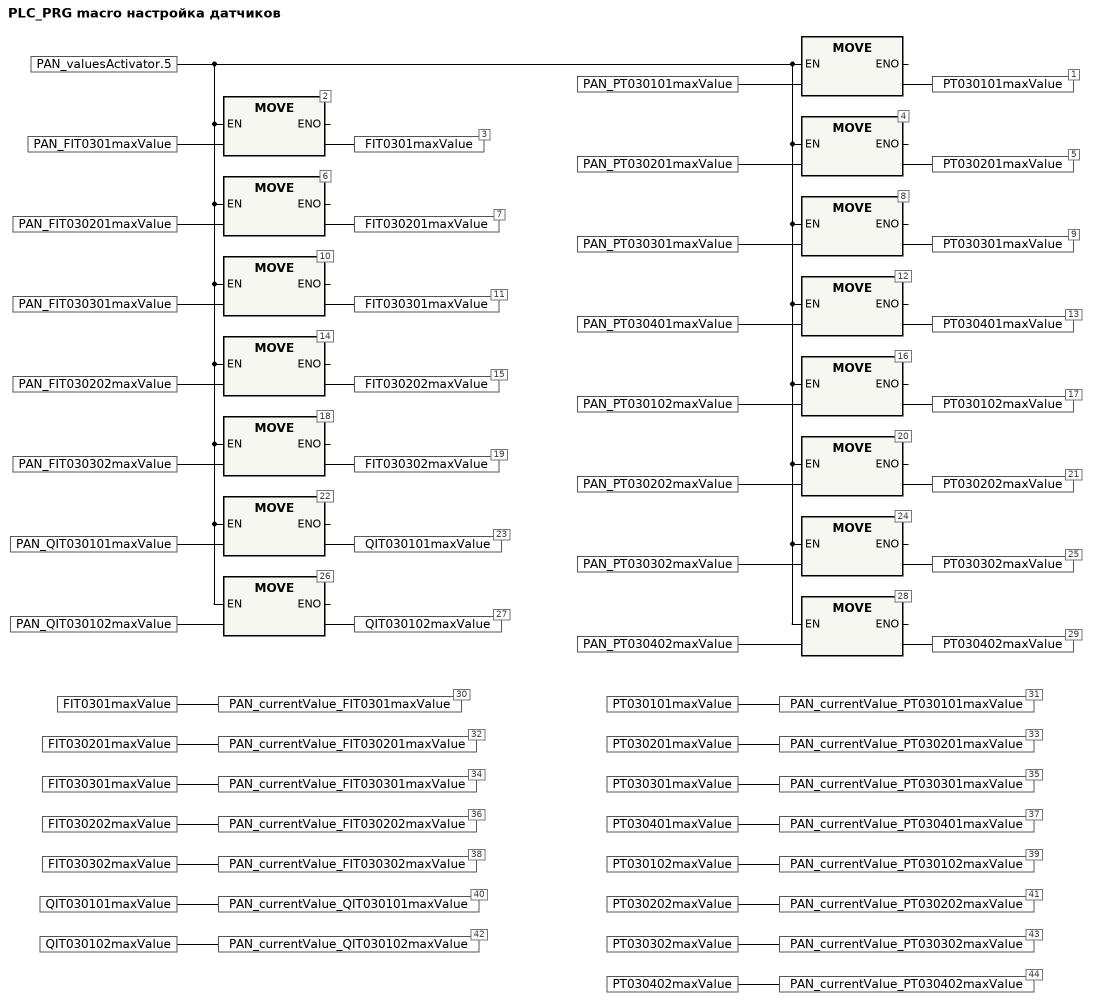
[picture p24: PLC_PRG macro настройка датчиков (CFC)]
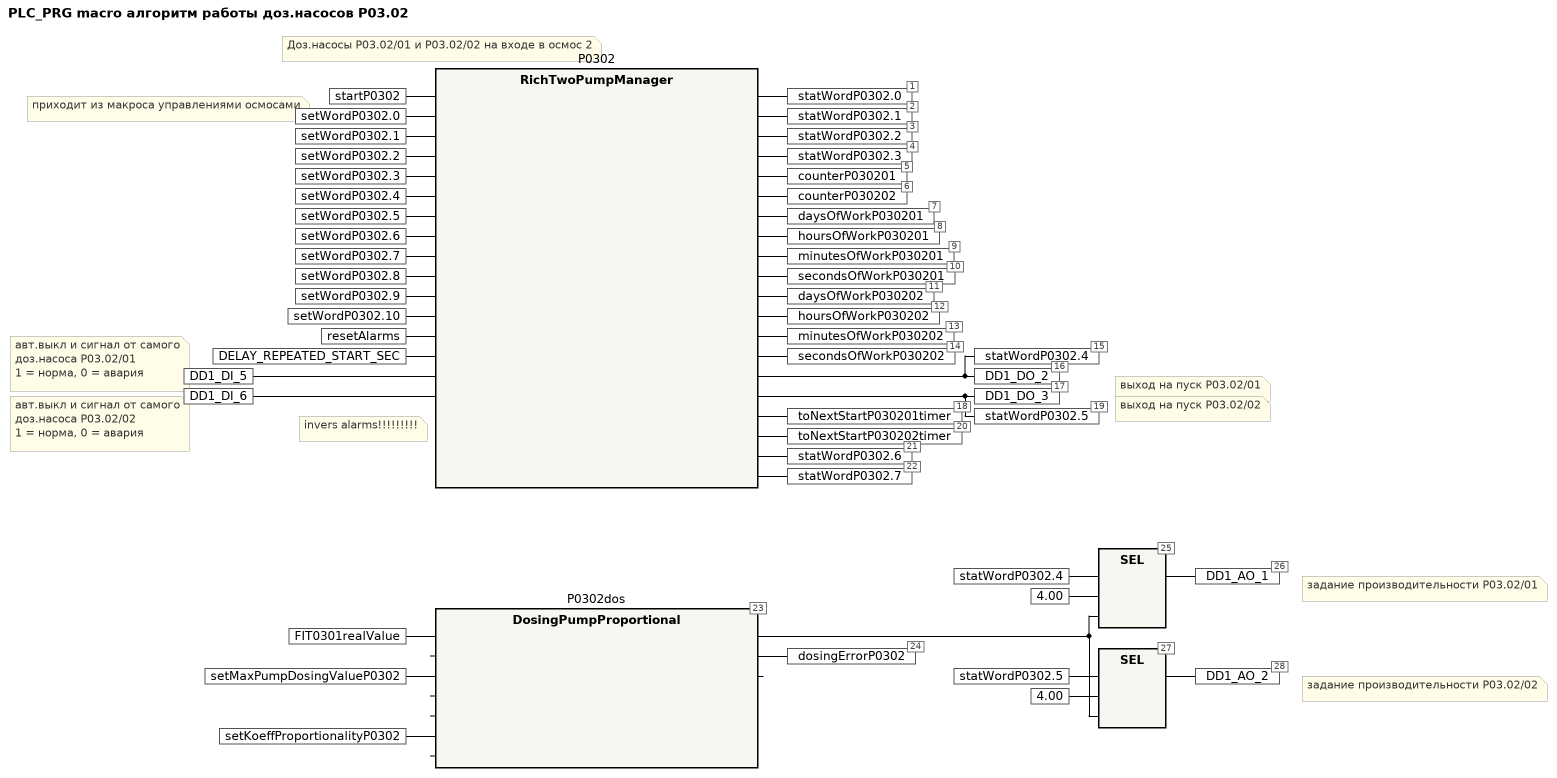
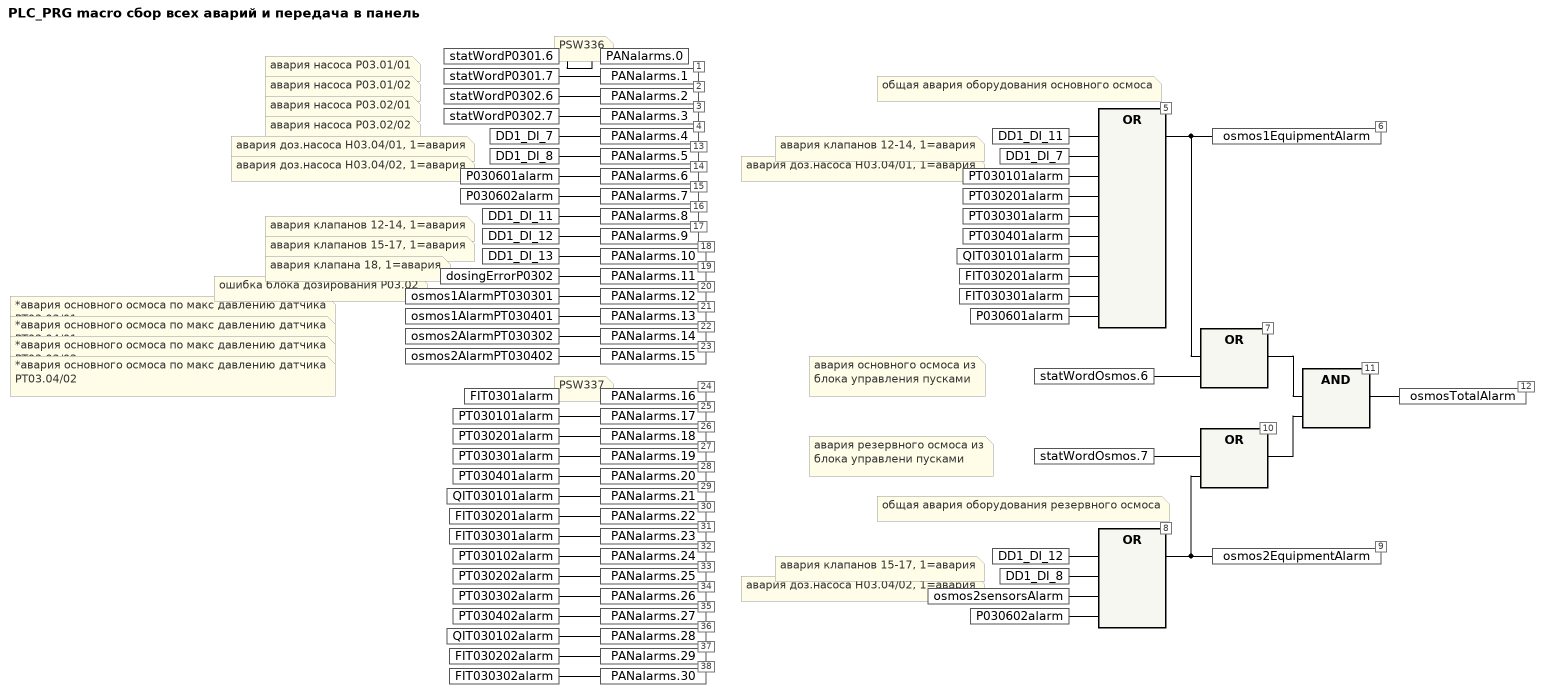
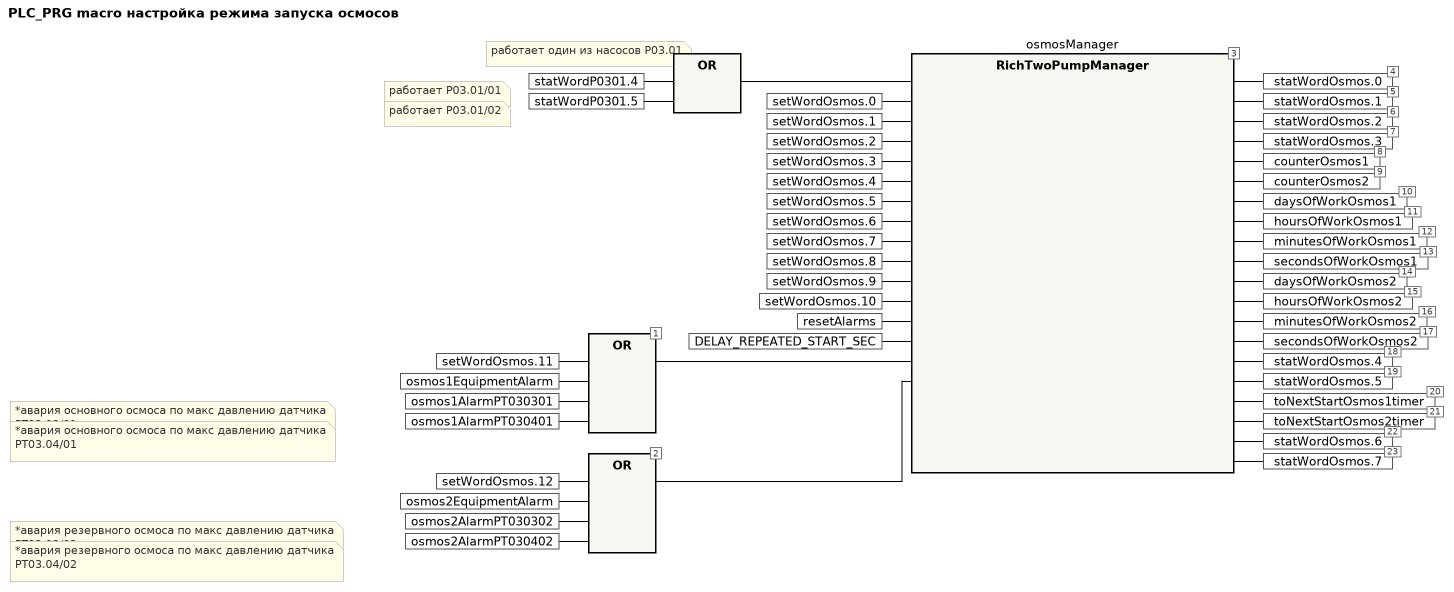
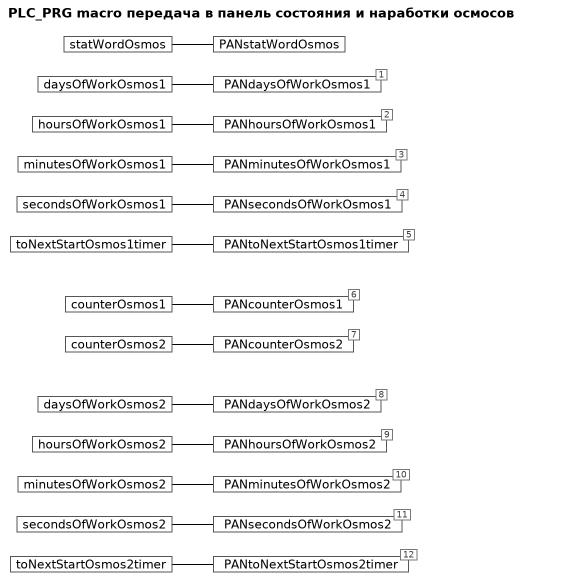
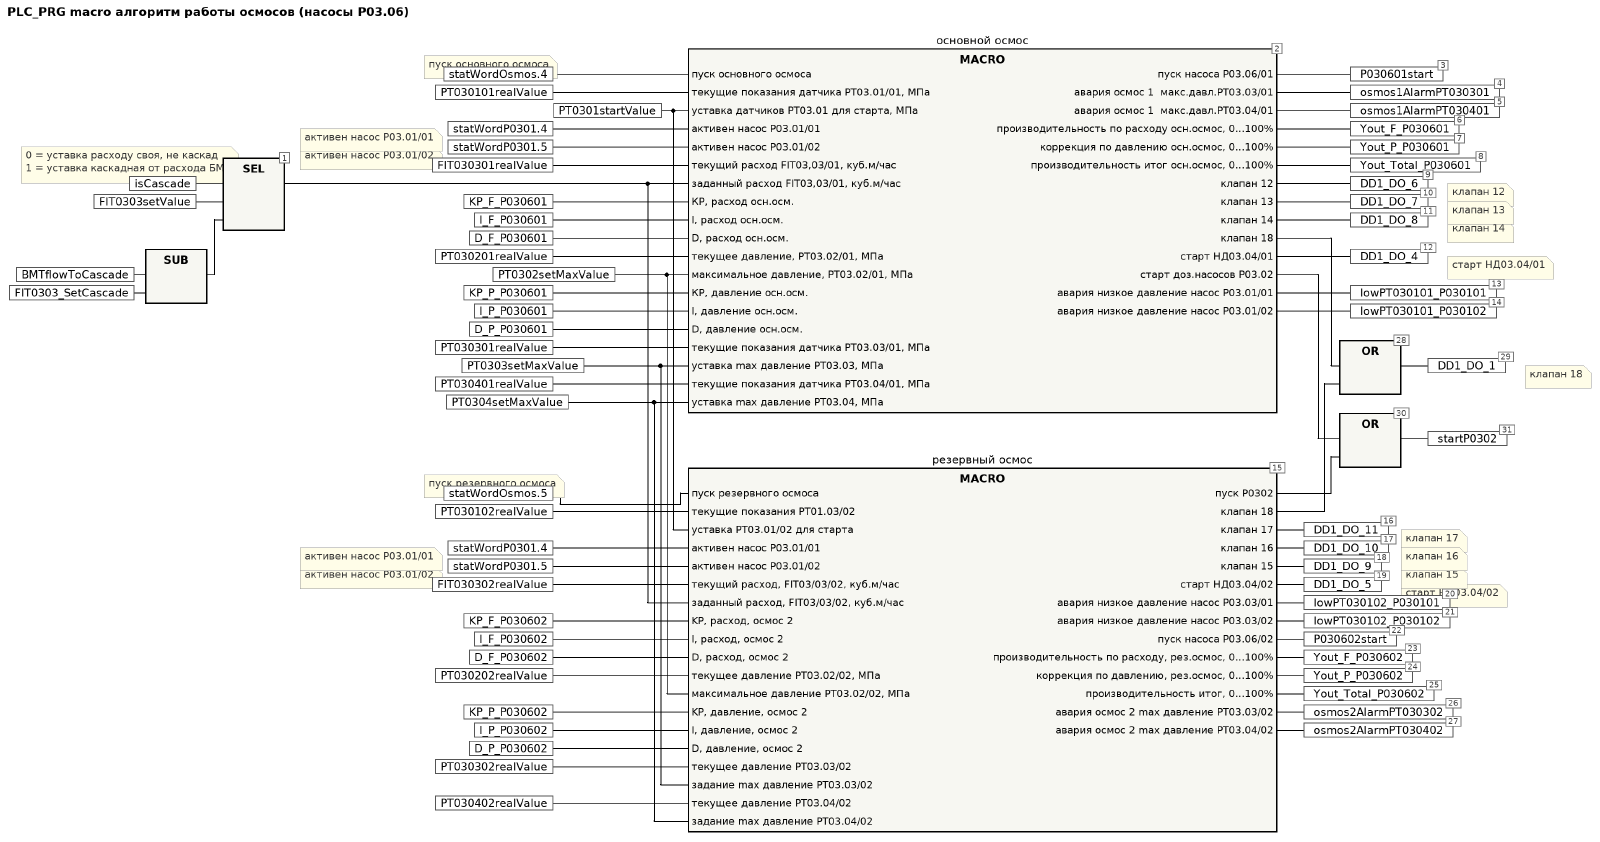
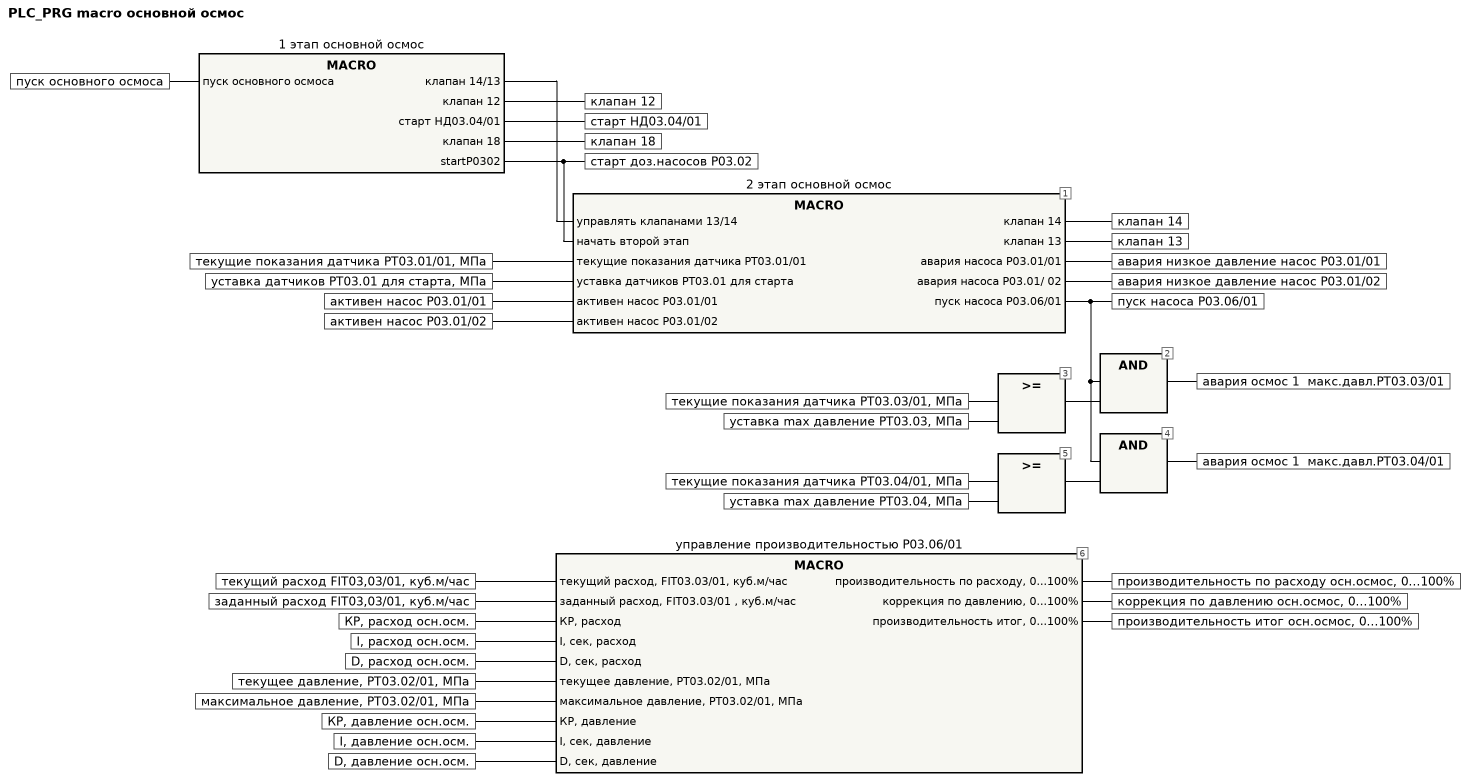
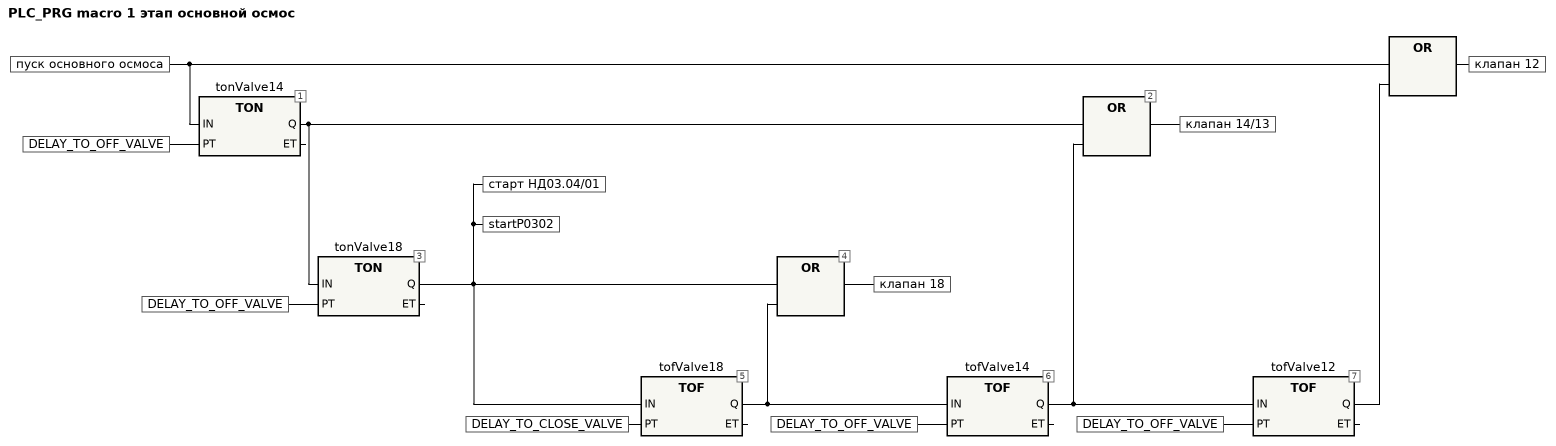
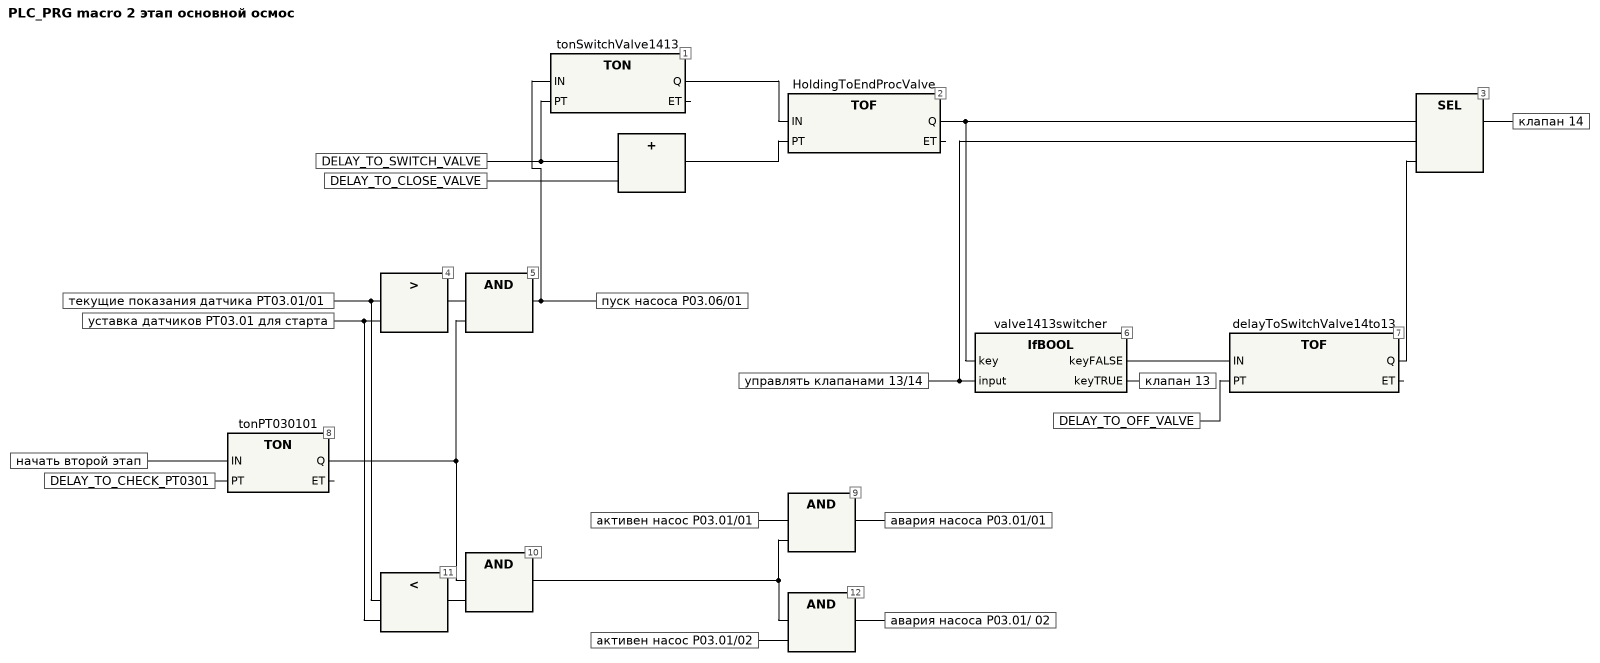
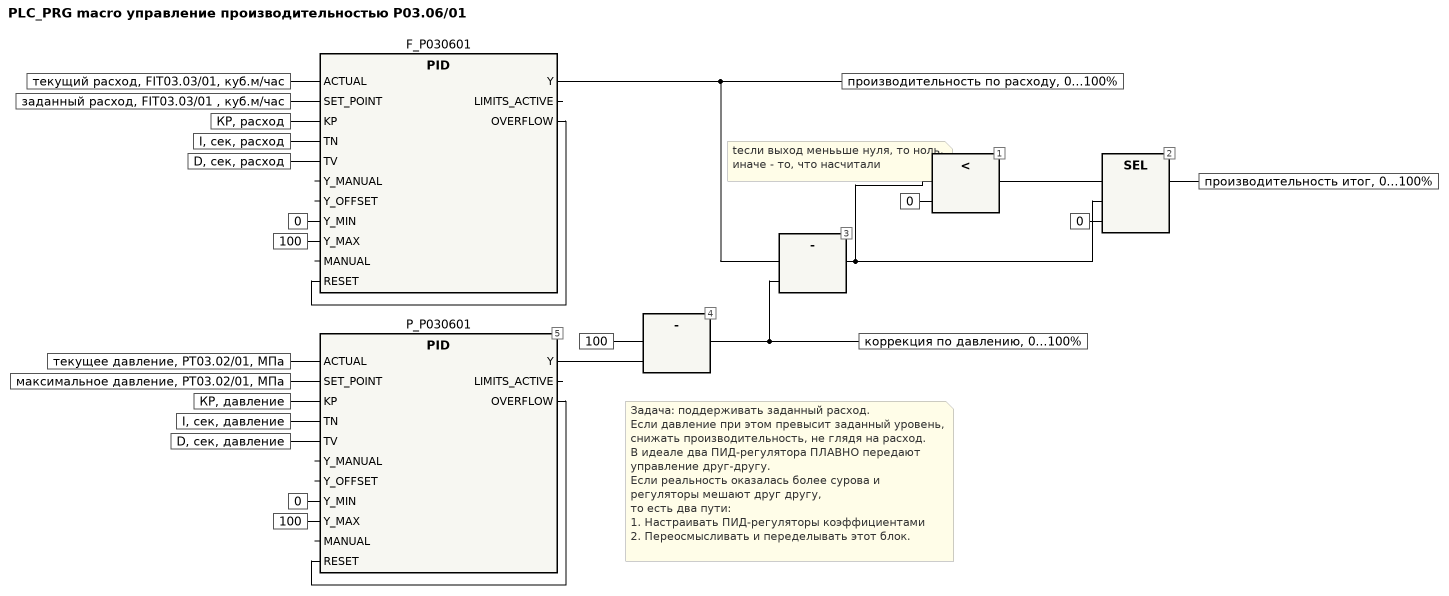
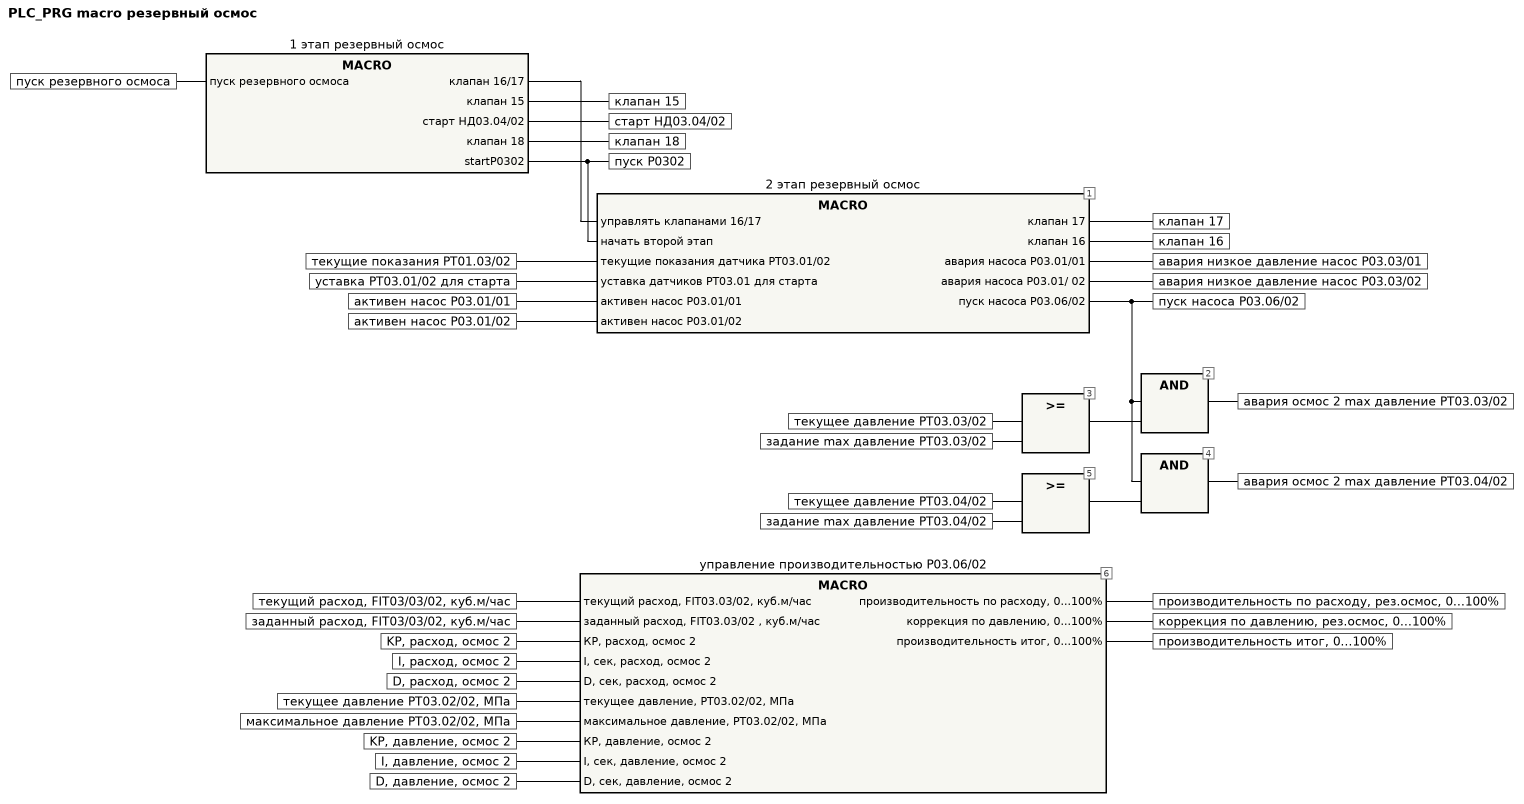
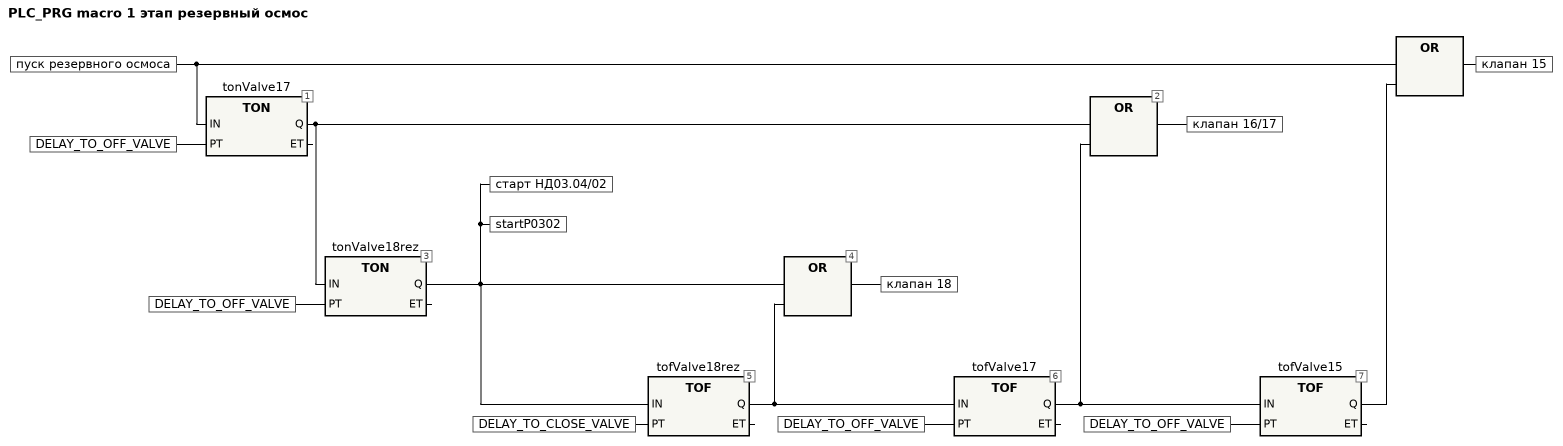
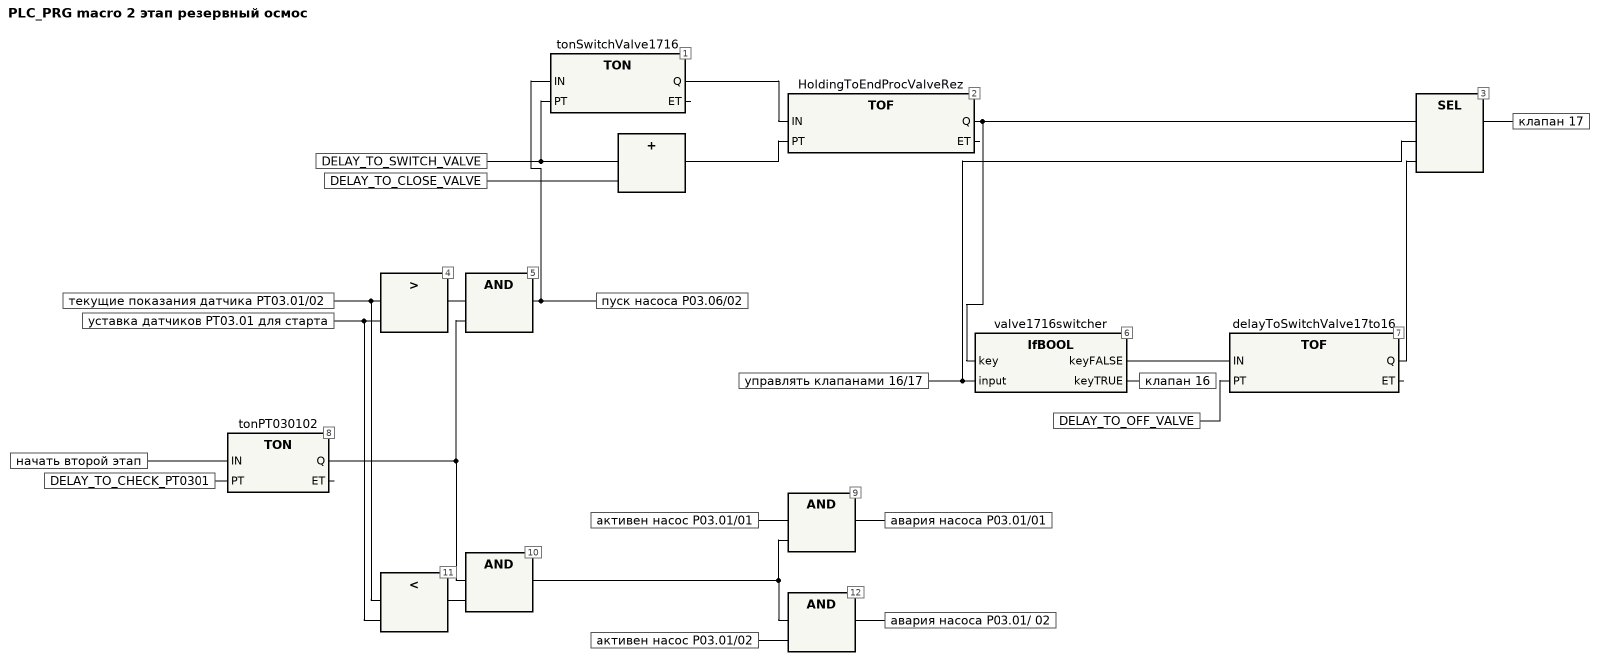
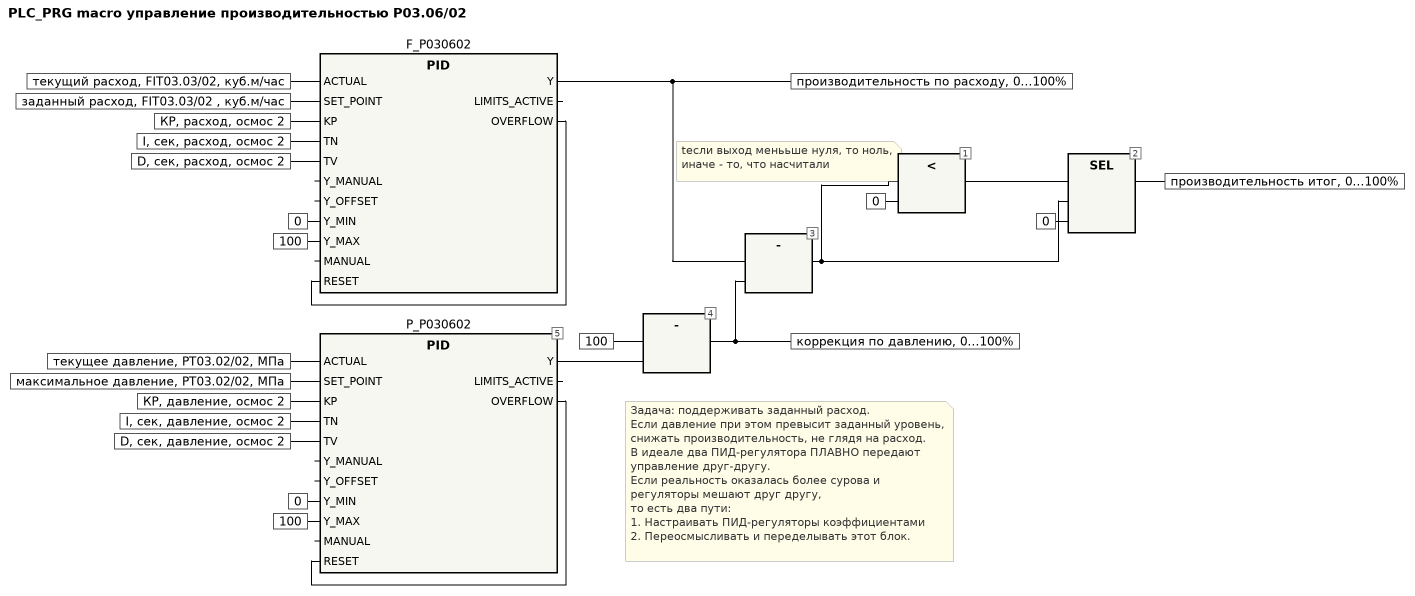
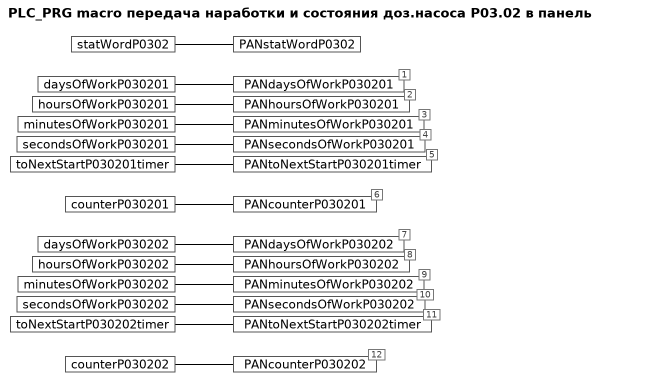
_CFC_ (* Continuous Function Chart, elements in execution order *)
(* восстановление заданного ранее режима / работы после подачи питания *)
(* командное слово удаленной панели *)
(* командное слово в локальной панели *)
(* - низкий уровень в емкости V02.07 / (сигнал из АСУ-2 осмос 1) 1 = true *)
(* - высокий уровень в емкости V06.01 / (сигнал из АСУ-1 общий) 1 = true *)
(* - высокий уровень в емкости V04.01 / (сигнал от БМТ, МЕ04) 1 = true *)
(* расход в БМТ для расчета каскадной уставки / получить из АСУ-1! *)
(* показ расхода БМТ в панели оператора *)
(* 0 = уставка расходу своя, не каскад / 1 = уставка каскадная от расхода БМТ *)
(* прием сигналов из разных источников / условие запуска см.в макросе "управление насосами Р03.01 *)
(* командное слово для осмоса *)
(* командное слово доз. насоса Р03.02 *)
(* командное слово насосов Р03.01 *)
(* PAN - переменные для панели в щите / OPAN - переменные для выносной панели, на установке *)
(* ******************добавь сюда вкл и выкл от выносной панели******************* / задание режима работы - каскад/не каскад *)
#0 onStartCatcher:R_TRIG(CLK: TRUE)
#1 OR(PANsetWordOsmos.11, #0.Q)
#2 resetAlarms <= #1
#3 setCascadeOnStart:IfBOOL(key: isCascadeOnStart, input: #0.Q)
#4 OR(#3.keyTRUE, PANsetWordOsmos.12)
#5 OR(#3.keyFALSE, PANsetWordOsmos.13)
#6 cascadeTrig:RS(SET: #4, RESET1: #5)
#7 statWordOsmos.8 <= #6.Q1
#8 isCascade <= #6.Q1
#9 MOVE(EN: #0.Q, setWordP0301onStart)
#10 setWordP0301 <= #9
#11 OR(#4, #5)
#12 MOVE(EN: #11, isCascade)
#13 isCascadeOnStart <= #12
#14 MOVE(EN: #0.Q, setWordP0302onStart)
#15 setWordP0302 <= #14
#16 MOVE(EN: #0.Q, setWordOsmosOnStart)
#17 setWordOsmos <= #16
#18 lowLevelV0207 <= ASU_Levels.0
#19 highLevelV0601 <= ASU_Levels.1
#20 highLevelV0401 <= ASU_Levels.2
#21 BMTflowToCascade <= ASU_FlowFromBMT
#22 PAN_BMT_Flow <= BMTflowToCascade
#23 MACRO настройка расхода, каскада и допустимых давлений осмоса()
	(* значение, вычитаемое из расхода БМТ / задается в панели, коэф.каскад *)
	(* предельно допустимые давления *)
	(* некаскадная уставка на поддержание расхода *)
	(* мин.давление для старта осмосов *)
	#24 MOVE(EN: PAN_valuesActivator.0, PAN_FIT0303_SetCascade)
	#25 FIT0303_SetCascade <= #24
	#26 MOVE(EN: PAN_valuesActivator.0, PAN_PT0301startValue)
	#27 PT0301startValue <= #26
	#28 MOVE(EN: PAN_valuesActivator.0, PAN_FIT0303setValue)
	#29 FIT0303setValue <= #28
	#30 MOVE(EN: PAN_valuesActivator.0, PAN_PT0302setMaxValue)
	#31 PT0302setMaxValue <= #30
	#32 MOVE(EN: PAN_valuesActivator.0, PAN_PT0303setMaxValue)
	#33 PT0303setMaxValue <= #32
	#34 MOVE(EN: PAN_valuesActivator.0, PAN_PT0304setMaxValue)
	#35 PT0304setMaxValue <= #34
	#36 PAN_currentValue_PT0301startValue <= PT0301startValue
	#37 PAN_currentValue_FIT0303setValue <= FIT0303setValue
	#38 PAN_currentValue_PT0302setMaxValue <= PT0302setMaxValue
	#39 PAN_currentValue_PT0303setMaxValue <= PT0303setMaxValue
	#40 PAN_currentValue_PT0304setMaxValue <= PT0304setMaxValue
	#41 PAN_currentValue_FIT0303_SetCascade <= FIT0303_SetCascade
END_MACRO
#42 MACRO коэффициенты ПИД-регуляторов осмосов()
	(* осмос 1 *)
	(* осмос 2 *)
	(* PID по расходу *)
	(* PID по давлению *)
	(* PID по расходу *)
	(* PID по давлению *)
	#43 MOVE(EN: PAN_valuesActivator.1, PAN_KP_F_P030601)
	#44 KP_F_P030601 <= #43
	#45 MOVE(EN: PAN_valuesActivator.1, PAN_I_F_P030601)
	#46 I_F_P030601 <= #45
	#47 MOVE(EN: PAN_valuesActivator.1, PAN_D_F_P030601)
	#48 D_F_P030601 <= #47
	#49 MOVE(EN: PAN_valuesActivator.1, PAN_KP_P_P030601)
	#50 KP_P_P030601 <= #49
	#51 MOVE(EN: PAN_valuesActivator.1, PAN_I_P_P030601)
	#52 I_P_P030601 <= #51
	#53 MOVE(EN: PAN_valuesActivator.1, PAN_D_P_P030601)
	#54 D_P_P030601 <= #53
	#55 MOVE(EN: PAN_valuesActivator.2, PAN_KP_F_P030602)
	#56 KP_F_P030602 <= #55
	#57 MOVE(EN: PAN_valuesActivator.2, PAN_I_F_P030602)
	#58 I_F_P030602 <= #57
	#59 MOVE(EN: PAN_valuesActivator.2, PAN_D_F_P030602)
	#60 D_F_P030602 <= #59
	#61 MOVE(EN: PAN_valuesActivator.2, PAN_KP_P_P030602)
	#62 KP_P_P030602 <= #61
	#63 MOVE(EN: PAN_valuesActivator.2, PAN_I_P_P030602)
	#64 I_P_P030602 <= #63
	#65 MOVE(EN: PAN_valuesActivator.2, PAN_D_P_P030602)
	#66 D_P_P030602 <= #65
	#67 PAN_currentValue_KP_F_P030601 <= KP_F_P030601
	#68 PAN_currentValue_KP_F_P030602 <= KP_F_P030602
	#69 PAN_currentValue_I_F_P030601 <= I_F_P030601
	#70 PAN_currentValue_I_F_P030602 <= I_F_P030602
	#71 PAN_currentValue_D_F_P030601 <= D_F_P030601
	#72 PAN_currentValue_D_F_P030602 <= D_F_P030602
	#73 PAN_currentValue_KP_P_P030601 <= KP_P_P030601
	#74 PAN_currentValue_KP_P_P030602 <= KP_P_P030602
	#75 PAN_currentValue_I_P_P030601 <= I_P_P030601
	#76 PAN_currentValue_I_P_P030602 <= I_P_P030602
	#77 PAN_currentValue_D_P_P030601 <= D_P_P030601
	#78 PAN_currentValue_D_P_P030602 <= D_P_P030602
END_MACRO
#79 MACRO обмен сигналами с DD2 (ПР102)()
	(* передача производительности / Р03.06/02 через модбас *)
	(* производительность доз.насоса Р03.06/02 / в процентах 0...100% *)
	(* 5430 - это число, соответствующее 100% / производительности ЧРП (50Гц) / так показали эксперименты в Казани / по РЭ и обучающим видео Овна 50Гц / соответствует число 16384 / Не знаю кому верить / Это число надо уточнить при ПНР... *)
	(* передача производительности / Р03.06/01 через модбас *)
	(* производительность доз.насоса Р03.06/01 / в процентах 0...100% *)
	(* сигнал на запуск Р03.06/02 *)
	(* получить из DD2 *)
	(* авария насоса Р03.06/02 *)
	(* передать в DD2 *)
	(* сигнал на запуск Р03.06/01 *)
	(* авария насоса Р03.06/01 *)
	(* есть авария хотя бы одного датчика в резеврном осмосе / получить из DD2 (ПР102), 1=авария *)
	(* сигнал на старт Р03.01/02 *)
	(* сигнал на старт Р03.01/01 *)
	#80 DO_bit_mask_DD2.0 <= statWordP0301.4
	#81 P030601alarm <= stat_word_P030601_PLC.3
	#82 DO_bit_mask_DD2.1 <= statWordP0301.5
	#83 P030602alarm <= stat_word_P030602_PLC.3
	#84 MACRO командное слово Р03.06/01(pin 1 "пуск/стоп": P030601start)
		(* не используется *)
		(* 0=набор 1, 1=набор 2 *)
		(* не используется *)
		(* 0=реле 1 выключено, 1=реле 1 включено *)
		(* 0=данные недействительны, 1=данные действительны *)
		(* 0=изменение скорости1 (согласно 3-4), 1=изменение скорости 2 (согласно 3-5) *)
		(* 0=работа по заданию, 1=фиксированная частота(параметр 3-11) *)
		(* 0=нет сброса, 1=сброс *)
		(* 0=останов с замедлением, 1=пуск *)
		(* фиксация частоты, 0=есть, 1=нет *)
		(* быстрый останов, 0=есть, 1=нет *)
		(* останов выбегом, 0=есть, 1=нет *)
		(* торможение постоянным током, 0=есть, 1=нет. *)
		(* предустановленное значение, старший бит, 0=0, 1=1 *)
		(* предустановленное значение, младший бит, 0=0, 1=1 *)
		#85 com_word_P030601_PLC.0 <= 0
		#86 com_word_P030601_PLC.1 <= 0
		#87 com_word_P030601_PLC.2 <= 1
		#88 com_word_P030601_PLC.3 <= pin 1
		#89 com_word_P030601_PLC.6 <= pin 1
		#90 com_word_P030601_PLC.4 <= 1
		#91 com_word_P030601_PLC.5 <= 1
		#92 com_word_P030601_PLC.7 <= 0
		#93 com_word_P030601_PLC.8 <= 0
		#94 com_word_P030601_PLC.9 <= 0
		#95 com_word_P030601_PLC.10 <= 1
		#96 com_word_P030601_PLC.11 <= 0
		#97 com_word_P030601_PLC.12 <= 0
		#98 com_word_P030601_PLC.13 <= 0
		#99 com_word_P030601_PLC.14 <= 0
	END_MACRO
	#100 MACRO командное слово Р03.06/02(pin 1 "пуск/стоп": P030602start)
		(* не используется *)
		(* 0=набор 1, 1=набор 2 *)
		(* не используется *)
		(* 0=реле 1 выключено, 1=реле 1 включено *)
		(* 0=данные недействительны, 1=данные действительны *)
		(* 0=изменение скорости1 (согласно 3-4), 1=изменение скорости 2 (согласно 3-5) *)
		(* 0=работа по заданию, 1=фиксированная частота(параметр 3-11) *)
		(* 0=нет сброса, 1=сброс *)
		(* 0=останов с замедлением, 1=пуск *)
		(* фиксация частоты, 0=есть, 1=нет *)
		(* быстрый останов, 0=есть, 1=нет *)
		(* останов выбегом, 0=есть, 1=нет *)
		(* торможение постоянным током, 0=есть, 1=нет. *)
		(* предустановленное значение, старший бит, 0=0, 1=1 *)
		(* предустановленное значение, младший бит, 0=0, 1=1 *)
		#101 com_word_P030602_PLC.0 <= 0
		#102 com_word_P030602_PLC.1 <= 0
		#103 com_word_P030602_PLC.2 <= 1
		#104 com_word_P030602_PLC.3 <= pin 1
		#105 com_word_P030602_PLC.6 <= pin 1
		#106 com_word_P030602_PLC.4 <= 1
		#107 com_word_P030602_PLC.5 <= 1
		#108 com_word_P030602_PLC.7 <= 0
		#109 com_word_P030602_PLC.8 <= 0
		#110 com_word_P030602_PLC.9 <= 0
		#111 com_word_P030602_PLC.10 <= 1
		#112 com_word_P030602_PLC.11 <= 0
		#113 com_word_P030602_PLC.12 <= 0
		#114 com_word_P030602_PLC.13 <= 0
		#115 com_word_P030602_PLC.14 <= 0
	END_MACRO
	#116 WORD_TO_BOOL(DI_bit_mask_DD2)
	#117 osmos2sensorsAlarm <= #116
	#118 freqP030601:LIN_TRAFO(IN: Yout_Total_P030601, IN_MIN: 0, IN_MAX: 100, OUT_MIN: 0, OUT_MAX: 16384)
	#119 REAL_TO_WORD(#118.OUT)
	#120 set_freq_P030601_PLC <= #119
	#121 MACRO обработка аналоговых сигналов DD2()
		(* Показания расходомера FIT03.01/01 на входе в осмос 2. / Для управления производительностью НД Р03.02 (1 и 2). *)
		(* давление датчик РТ03.01/02 *)
		(* давление датчик РТ03.02/02 *)
		(* давление датчик РТ03.03/02 *)
		(* давление датчик РТ03.04/02 *)
		(* расходомер FIT03.03/02 *)
		(* расходомер FIT03.02/02 *)
		(* кондуктомер QIT03.01/02 *)
		#122 pt030102:ControlAI(PT030102rawValue, -, PT030102maxValue)
		#123 PT030102realValue <= #122.out 1
		#124 PT030102alarm <= #122.out 2
		#125 pt030202:ControlAI(PT030202rawValue, -, PT030202maxValue)
		#126 PT030202realValue <= #125.out 1
		#127 PT030202alarm <= #125.out 2
		#128 pt030302:ControlAI(PT030302rawValue, -, PT030302maxValue)
		#129 PT030302realValue <= #128.out 1
		#130 PT030302alarm <= #128.out 2
		#131 pt030402:ControlAI(PT030402rawValue, -, PT030402maxValue)
		#132 PT030402realValue <= #131.out 1
		#133 PT030402alarm <= #131.out 2
		#134 fit0301:ControlAI(FIT030101rawValue, -, FIT0301maxValue)
		#135 FIT0301realValue <= #134.out 1
		#136 FIT0301alarm <= #134.out 2
		#137 fit030202:ControlAI(FIT030202rawValue, -, FIT030202maxValue)
		#138 FIT030202realValue <= #137.out 1
		#139 FIT030202alarm <= #137.out 2
		#140 fit030302:ControlAI(FIT030302rawValue, -, FIT030302maxValue)
		#141 FIT030302realValue <= #140.out 1
		#142 FIT030302alarm <= #140.out 2
		#143 qit030102:ControlAI(QIT030102rawValue, -, QIT030102maxValue)
		#144 QIT030102realValue <= #143.out 1
		#145 QIT030102alarm <= #143.out 2
	END_MACRO
	#146 freqP030602:LIN_TRAFO(IN: Yout_Total_P030602, IN_MIN: 0, IN_MAX: 100, OUT_MIN: 0, OUT_MAX: 16384)
	#147 REAL_TO_WORD(#146.OUT)
	#148 set_freq_P030602_PLC <= #147
END_MACRO
#149 MACRO передача наработки и состояния насосов Р03.01 в панель()
	#150 PANstatWordP0301 <= statWordP0301
	#151 PANdaysOfWorkP030101 <= daysOfWorkP030101
	#152 PANhoursOfWorkP030101 <= hoursOfWorkP030101
	#153 PANminutesOfWorkP030101 <= minutesOfWorkP030101
	#154 PANsecondsOfWorkP030101 <= secondsOfWorkP030101
	#155 PANtoNextStartP030101timer <= toNextStartP030101timer
	#156 PANcounterP030101 <= counterP030101
	#157 PANdaysOfWorkP030102 <= daysOfWorkP030102
	#158 PANhoursOfWorkP030102 <= hoursOfWorkP030102
	#159 PANminutesOfWorkP030102 <= minutesOfWorkP030102
	#160 PANsecondsOfWorkP030102 <= secondsOfWorkP030102
	#161 PANtoNextStartP030102timer <= toNextStartP030102timer
	#162 PANcounterP030102 <= counterP030102
END_MACRO
#163 WORD_TO_BOOL(PANsetWordP0301)
#164 tof1:TOF(IN: #163, PT: T#1s)
#165 MOVE(EN: #164.Q, PANsetWordP0301)
#166 setWordP0301 <= #165
#167 WORD_TO_BOOL(OPANsetWordP0301)
#168 tof2:TOF(IN: #167, PT: T#1s)
#169 OR(#164.Q, #168.Q)
#170 MOVE(EN: #169, statWordP0301)
#171 setWordP0301onStart <= #170
#172 MOVE(EN: #168.Q, OPANsetWordP0301)
#173 setWordP0301 <= #172
#174 MACRO уставки доз.насосов Р03.02()
	(* max производительность доз.насоса Р03.02 *)
	(* задание дозирования, мл/куб.м *)
	#175 MOVE(EN: PAN_valuesActivator.3, PANsetMaxPumpDosingValueP0302)
	#176 setMaxPumpDosingValueP0302 <= #175
	#177 MOVE(EN: PAN_valuesActivator.3, PANsetKoeffPropotrionalityP0302)
	#178 setKoeffProportionalityP0302 <= #177
	#179 PAN_currentValue_setMaxPumpDosingValueP0302 <= setMaxPumpDosingValueP0302
	#180 PAN_currentValue_setKoeffProportionalityP0302 <= setKoeffProportionalityP0302
END_MACRO
#181 MACRO обработка аналоговых сигналов датчиков основного осмоса()
	#182 controlAIpt030101:ControlAI(DD1_AI_2, -, PT030101maxValue)
	#183 PT030101realValue <= #182.out 1
	#184 PT030101alarm <= #182.out 2
	#185 controlAIpt030201:ControlAI(DD1_AI_3, -, PT030201maxValue)
	#186 PT030201realValue <= #185.out 1
	#187 PT030201alarm <= #185.out 2
	#188 controlAIpt030301:ControlAI(DD1_AI_4, -, PT030301maxValue)
	#189 PT030301realValue <= #188.out 1
	#190 PT030301alarm <= #188.out 2
	#191 controlAIpt030401:ControlAI(DD1_AI_5, -, PT030401maxValue)
	#192 PT030401realValue <= #191.out 1
	#193 PT030401alarm <= #191.out 2
	#194 controlAIqit030101:ControlAI(DD1_AI_6, -, QIT030101maxValue)
	#195 QIT030101realValue <= #194.out 1
	#196 QIT030101alarm <= #194.out 2
	#197 controlAIfit030201:ControlAI(DD1_AI_7, -, FIT030201maxValue)
	#198 FIT030201realValue <= #197.out 1
	#199 FIT030201alarm <= #197.out 2
	#200 controlAIfit030301:ControlAI(DD1_AI_8, -, FIT030301maxValue)
	#201 FIT030301realValue <= #200.out 1
	#202 FIT030301alarm <= #200.out 2
END_MACRO
#203 MACRO передача показаний датчиков в панель оператора()
	#204 PAN_FIT0301realValue <= FIT0301realValue
	#205 PAN_PT030101realValue <= PT030101realValue
	#206 PAN_PT030201realValue <= PT030201realValue
	#207 PAN_PT030301realValue <= PT030301realValue
	#208 PAN_FIT030301realValue <= FIT030301realValue
	#209 PAN_PT030102realValue <= PT030102realValue
	#210 PAN_PT030202realValue <= PT030202realValue
	#211 PAN_PT030302realValue <= PT030302realValue
	#212 PAN_FIT030302realValue <= FIT030302realValue
	#213 PAN_PT030401realValue <= PT030401realValue
	#214 PAN_FIT030201realValue <= FIT030201realValue
	#215 PAN_QIT030101realValue <= QIT030101realValue
	#216 PAN_PT030402realValue <= PT030402realValue
	#217 PAN_FIT030202realValue <= FIT030202realValue
	#218 PAN_QIT030102realValue <= QIT030102realValue
END_MACRO
#219 MACRO задание задержек времени из панели()
	(* задержка до переключения клапанов после запуска Р0306 *)
	(* задержка перед открытием/закрытием клапанов при / последовательном открытии/закрытии при старте осмоса *)
	(* время задержки начала контроля параметра (например, задержка / контроля эк.манометра после насоса, время на разгон). *)
	(* Время задержки повторного пуска насосов, сек *)
	(* задержка контроля датчика РТ0301 *)
	(* задержка до начала закрытия клапанов после выключения насоса *)
	(* T#5s *)
	(* 15 *)
	(* T#3s *)
	(* T#10s *)
	(* T#15s *)
	(* T#10s *)
	#220 MACRO word to time(pin 1 "word_in": PAN_CHECKING_DELAY_TIME)
		#221 UINT_TO_UDINT(pin 1)
		#222 MUL(#221, 1000)
		#223 UDINT_TO_TIME(#222)
		out 1 "time_out" <= #223
	END_MACRO
	#224 MOVE(EN: PAN_valuesActivator.4, #220.out 1)
	#225 CHECKING_DELAY_TIME <= #224
	#226 MOVE(EN: PAN_valuesActivator.4, PAN_DELAY_REPEATED_START_SEC)
	#227 DELAY_REPEATED_START_SEC <= #226
	#228 MACRO word to time(pin 1 "word_in": PAN_DELAY_TO_OFF_VALVE)
		#229 UINT_TO_UDINT(pin 1)
		#230 MUL(#229, 1000)
		#231 UDINT_TO_TIME(#230)
		out 1 "time_out" <= #231
	END_MACRO
	#232 MOVE(EN: PAN_valuesActivator.4, #228.out 1)
	#233 DELAY_TO_OFF_VALVE <= #232
	#234 MACRO word to time(pin 1 "word_in": PAN_DELAY_TO_CHECK_PT0301)
		#235 UINT_TO_UDINT(pin 1)
		#236 MUL(#235, 1000)
		#237 UDINT_TO_TIME(#236)
		out 1 "time_out" <= #237
	END_MACRO
	#238 MOVE(EN: PAN_valuesActivator.4, #234.out 1)
	#239 DELAY_TO_CHECK_PT0301 <= #238
	#240 MACRO word to time(pin 1 "word_in": PAN_DELAY_TO_SWITCH_VALVE)
		#241 UINT_TO_UDINT(pin 1)
		#242 MUL(#241, 1000)
		#243 UDINT_TO_TIME(#242)
		out 1 "time_out" <= #243
	END_MACRO
	#244 MOVE(EN: PAN_valuesActivator.4, #240.out 1)
	#245 DELAY_TO_SWITCH_VALVE <= #244
	#246 MACRO word to time(pin 1 "word_in": PAN_DELAY_TO_CLOSE_VALVE)
		#247 UINT_TO_UDINT(pin 1)
		#248 MUL(#247, 1000)
		#249 UDINT_TO_TIME(#248)
		out 1 "time_out" <= #249
	END_MACRO
	#250 MOVE(EN: PAN_valuesActivator.4, #246.out 1)
	#251 DELAY_TO_CLOSE_VALVE <= #250
	#252 MACRO time to word(pin 1 "time_in": CHECKING_DELAY_TIME)
		#253 TIME_TO_UDINT(pin 1)
		#254 DIV(#253, 1000)
		#255 UDINT_TO_UINT(#254)
		out 1 "uint_out" <= #255
	END_MACRO
	#256 PAN_currentValue_CHECKING_DELAY_TIME <= #252.out 1
	#257 PAN_currentValue_DELAY_REPEATED_START_SEC <= DELAY_REPEATED_START_SEC
	#258 MACRO time to word(pin 1 "time_in": DELAY_TO_OFF_VALVE)
		#259 TIME_TO_UDINT(pin 1)
		#260 DIV(#259, 1000)
		#261 UDINT_TO_UINT(#260)
		out 1 "uint_out" <= #261
	END_MACRO
	#262 PAN_currentValue_DELAY_TO_OFF_VALVE <= #258.out 1
	#263 MACRO time to word(pin 1 "time_in": DELAY_TO_CHECK_PT0301)
		#264 TIME_TO_UDINT(pin 1)
		#265 DIV(#264, 1000)
		#266 UDINT_TO_UINT(#265)
		out 1 "uint_out" <= #266
	END_MACRO
	#267 PAN_currentValue_DELAY_TO_CHECK_PT0301 <= #263.out 1
	#268 MACRO time to word(pin 1 "time_in": DELAY_TO_SWITCH_VALVE)
		#269 TIME_TO_UDINT(pin 1)
		#270 DIV(#269, 1000)
		#271 UDINT_TO_UINT(#270)
		out 1 "uint_out" <= #271
	END_MACRO
	#272 PAN_currentValue_DELAY_TO_SWITCH_VALVE <= #268.out 1
	#273 MACRO time to word(pin 1 "time_in": DELAY_TO_CLOSE_VALVE)
		#274 TIME_TO_UDINT(pin 1)
		#275 DIV(#274, 1000)
		#276 UDINT_TO_UINT(#275)
		out 1 "uint_out" <= #276
	END_MACRO
	#277 PAN_currentValue_DELAY_TO_CLOSE_VALVE <= #273.out 1
END_MACRO
#278 MACRO управление насосами Р03.01 на входе в осмос()
	(* сигнал на пуск Р03.01/02 *)
	(* сигнал на пуск Р03.01/01 *)
	(* условие на запуск осмоса *)
	(* авария обоих осмосов, 1 = авария *)
	(* авария клапана 18, 1 = авария *)
	(* авария обоих доз. насосов / Р03.02 на входе в осмос, 1 = авария *)
	(* насосы Р03.01/01 и Р03.01/02 на входе в осмос / работают если нет: / - низкий уровень в емкости V02.07 = false / - высокий уровень в емкости V06.01 = false / - высокий уровень в емкости V04.01 (БМТ) = false *)
	(* - низкий уровень в емкости V02.07 / (сигнал из АСУ-2 осмос 1) 1 = true *)
	(* - высокий уровень в емкости V06.01 / (сигнал из АСУ-1 общий) 1 = true *)
	(* - высокий уровень в емкости V04.01 / (сигнал от БМТ, МЕ04) 1 = true *)
	(* авария Р03.01/01 *)
	(* автомат Р03.01/01, 1 = норма / 0 = авария *)
	(* сигнал на пуск Р03.01/01 *)
	(* автомат Р03.01/02, 1 = норма / 0 = авария *)
	(* э.к.манометр Р03.01/01 / 1 = норма / 0 = нет давления *)
	(* э.к.манометр Р03.01/02 / 1 = норма / 0 = нет давления *)
	(* сигнал на пуск Р03.01/02 *)
	(* авария Р03.01/02 *)
	#279 AND(NOT lowLevelV0207, NOT highLevelV0601, NOT highLevelV0401)
	#280 AND(NOT alarmP0302, NOT DD1_DI_13, NOT osmosTotalAlarm)
	#281 AND(#279, #280)
	#282 P0301:RichTwoPumpManager(#281, setWordP0301.0, setWordP0301.1, setWordP0301.2, setWordP0301.3, setWordP0301.4, setWordP0301.5, setWordP0301.6, setWordP0301.7, setWordP0301.8, setWordP0301.9, setWordP0301.10, resetAlarms, DELAY_REPEATED_START_SEC, alarmP030101, alarmP030102)
	#283 statWordP0301.0 <= #282.out 1
	#284 statWordP0301.1 <= #282.out 2
	#285 statWordP0301.2 <= #282.out 3
	#286 statWordP0301.3 <= #282.out 4
	#287 counterP030101 <= #282.out 5
	#288 counterP030102 <= #282.out 6
	#289 daysOfWorkP030101 <= #282.out 7
	#290 hoursOfWorkP030101 <= #282.out 8
	#291 minutesOfWorkP030101 <= #282.out 9
	#292 secondsOfWorkP030101 <= #282.out 10
	#293 daysOfWorkP030102 <= #282.out 11
	#294 hoursOfWorkP030102 <= #282.out 12
	#295 minutesOfWorkP030102 <= #282.out 13
	#296 secondsOfWorkP030102 <= #282.out 14
	#297 statWordP0301.4 <= #282.out 15
	#298 statWordP0301.5 <= #282.out 16
	#299 toNextStartP030101timer <= #282.out 17
	#300 toNextStartP030102timer <= #282.out 18
	#301 statWordP0301.6 <= #282.out 19
	#302 statWordP0301.7 <= #282.out 20
	#303 delayCheckIfP030102works:TON(IN: statWordP0301.5, PT: CHECKING_DELAY_TIME)
	#304 AND(NOT DD1_DI_4, #303.Q)
	#305 OR(NOT DD1_DI_2, lowPT030101_P030102, lowPT030102_P030102, #304)
	#306 alarmP030102 <= #305
	#307 delayCheckIfP030101works:TON(IN: statWordP0301.4, PT: CHECKING_DELAY_TIME)
	#308 AND(NOT DD1_DI_3, #307.Q)
	#309 OR(NOT DD1_DI_1, lowPT030101_P030101, lowPT030102_P030101, #308)
	#310 alarmP030101 <= #309
END_MACRO
#311 MACRO передача на главный экран панели статусов работы()
	(* valve 18 *)
	(* valve 17 *)
	(* valve 16 *)
	(* valve 15 *)
	(* valve 14 *)
	(* valve 13 *)
	(* valve 12 *)
	(* P03.04/02 *)
	(* P03.04/01 *)
	(* PIS03.01/02 *)
	(* PIS03.01/01 *)
	#312 PANmainViewBools.0 <= DD1_DI_3
	#313 PANmainViewBools.1 <= DD1_DI_4
	#314 PANmainViewBools.2 <= DD1_DO_4
	#315 PANmainViewBools.3 <= DD1_DO_5
	#316 PANmainViewBools.4 <= P030601start
	#317 PANmainViewBools.5 <= P030602start
	#318 PANmainViewBools.6 <= DD1_DO_6
	#319 PANmainViewBools.7 <= DD1_DO_7
	#320 PANmainViewBools.8 <= DD1_DO_8
	#321 PANmainViewBools.9 <= DD1_DO_9
	#322 PANmainViewBools.10 <= DD1_DO_10
	#323 PANmainViewBools.11 <= DD1_DO_11
	#324 PANmainViewBools.12 <= DD1_DO_1
	#325 PANmainViewBools.13 <= NOT lowLevelV0207
	#326 PANmainViewBools.14 <= NOT highLevelV0601
	#327 PANmainViewBools.15 <= NOT highLevelV0401
END_MACRO
#328 MACRO настройка датчиков()
	#329 MOVE(EN: PAN_valuesActivator.5, PAN_PT030101maxValue)
	#330 PT030101maxValue <= #329
	#331 MOVE(EN: PAN_valuesActivator.5, PAN_FIT0301maxValue)
	#332 FIT0301maxValue <= #331
	#333 MOVE(EN: PAN_valuesActivator.5, PAN_PT030201maxValue)
	#334 PT030201maxValue <= #333
	#335 MOVE(EN: PAN_valuesActivator.5, PAN_FIT030201maxValue)
	#336 FIT030201maxValue <= #335
	#337 MOVE(EN: PAN_valuesActivator.5, PAN_PT030301maxValue)
	#338 PT030301maxValue <= #337
	#339 MOVE(EN: PAN_valuesActivator.5, PAN_FIT030301maxValue)
	#340 FIT030301maxValue <= #339
	#341 MOVE(EN: PAN_valuesActivator.5, PAN_PT030401maxValue)
	#342 PT030401maxValue <= #341
	#343 MOVE(EN: PAN_valuesActivator.5, PAN_FIT030202maxValue)
	#344 FIT030202maxValue <= #343
	#345 MOVE(EN: PAN_valuesActivator.5, PAN_PT030102maxValue)
	#346 PT030102maxValue <= #345
	#347 MOVE(EN: PAN_valuesActivator.5, PAN_FIT030302maxValue)
	#348 FIT030302maxValue <= #347
	#349 MOVE(EN: PAN_valuesActivator.5, PAN_PT030202maxValue)
	#350 PT030202maxValue <= #349
	#351 MOVE(EN: PAN_valuesActivator.5, PAN_QIT030101maxValue)
	#352 QIT030101maxValue <= #351
	#353 MOVE(EN: PAN_valuesActivator.5, PAN_PT030302maxValue)
	#354 PT030302maxValue <= #353
	#355 MOVE(EN: PAN_valuesActivator.5, PAN_QIT030102maxValue)
	#356 QIT030102maxValue <= #355
	#357 MOVE(EN: PAN_valuesActivator.5, PAN_PT030402maxValue)
	#358 PT030402maxValue <= #357
	#359 PAN_currentValue_FIT0301maxValue <= FIT0301maxValue
	#360 PAN_currentValue_PT030101maxValue <= PT030101maxValue
	#361 PAN_currentValue_FIT030201maxValue <= FIT030201maxValue
	#362 PAN_currentValue_PT030201maxValue <= PT030201maxValue
	#363 PAN_currentValue_FIT030301maxValue <= FIT030301maxValue
	#364 PAN_currentValue_PT030301maxValue <= PT030301maxValue
	#365 PAN_currentValue_FIT030202maxValue <= FIT030202maxValue
	#366 PAN_currentValue_PT030401maxValue <= PT030401maxValue
	#367 PAN_currentValue_FIT030302maxValue <= FIT030302maxValue
	#368 PAN_currentValue_PT030102maxValue <= PT030102maxValue
	#369 PAN_currentValue_QIT030101maxValue <= QIT030101maxValue
	#370 PAN_currentValue_PT030202maxValue <= PT030202maxValue
	#371 PAN_currentValue_QIT030102maxValue <= QIT030102maxValue
	#372 PAN_currentValue_PT030302maxValue <= PT030302maxValue
	#373 PAN_currentValue_PT030402maxValue <= PT030402maxValue
END_MACRO
#374 MACRO алгоритм работы доз.насосов Р03.02()
	(* приходит из макроса управлениями осмосами *)
	(* авт.выкл и сигнал от самого / доз.насоса Р03.02/02 / 1 = норма, 0 = авария *)
	(* авт.выкл и сигнал от самого / доз.насоса Р03.02/01 / 1 = норма, 0 = авария *)
	(* Доз.насосы Р03.02/01 и Р03.02/02 на входе в осмос 2 *)
	(* выход на пуск Р03.02/01 *)
	(* задание производительности Р03.02/01 *)
	(* задание производительности Р03.02/02 *)
	(* выход на пуск Р03.02/02 *)
	(* invers alarms!!!!!!!!! *)
	#375 P0302:RichTwoPumpManager(startP0302, setWordP0302.0, setWordP0302.1, setWordP0302.2, setWordP0302.3, setWordP0302.4, setWordP0302.5, setWordP0302.6, setWordP0302.7, setWordP0302.8, setWordP0302.9, setWordP0302.10, resetAlarms, DELAY_REPEATED_START_SEC, DD1_DI_5, DD1_DI_6)
	#376 statWordP0302.0 <= #375.out 1
	#377 statWordP0302.1 <= #375.out 2
	#378 statWordP0302.2 <= #375.out 3
	#379 statWordP0302.3 <= #375.out 4
	#380 counterP030201 <= #375.out 5
	#381 counterP030202 <= #375.out 6
	#382 daysOfWorkP030201 <= #375.out 7
	#383 hoursOfWorkP030201 <= #375.out 8
	#384 minutesOfWorkP030201 <= #375.out 9
	#385 secondsOfWorkP030201 <= #375.out 10
	#386 daysOfWorkP030202 <= #375.out 11
	#387 hoursOfWorkP030202 <= #375.out 12
	#388 minutesOfWorkP030202 <= #375.out 13
	#389 secondsOfWorkP030202 <= #375.out 14
	#390 statWordP0302.4 <= #375.out 15
	#391 DD1_DO_2 <= #375.out 15
	#392 DD1_DO_3 <= #375.out 16
	#393 toNextStartP030201timer <= #375.out 17
	#394 statWordP0302.5 <= #375.out 16
	#395 toNextStartP030202timer <= #375.out 18
	#396 statWordP0302.6 <= #375.out 19
	#397 statWordP0302.7 <= #375.out 20
	#398 P0302dos:DosingPumpProportional(FIT0301realValue, -, setMaxPumpDosingValueP0302, -, -, setKoeffProportionalityP0302, -)
	#399 dosingErrorP0302 <= #398.out 2
	#400 SEL(statWordP0302.4, 4.00, #398.out 1)
	#401 DD1_AO_1 <= #400
	#402 SEL(statWordP0302.5, 4.00, #398.out 1)
	#403 DD1_AO_2 <= #402
END_MACRO
#404 MACRO сбор всех аварий и передача в панель()
	(* авария доз.насоса Н03.04/02, 1=авария *)
	(* общая авария оборудования резервного осмоса *)
	(* авария клапанов 15-17, 1=авария *)
	(* общая авария оборудования основного осмоса *)
	(* авария доз.насоса Н03.04/01, 1=авария *)
	(* авария клапанов 12-14, 1=авария *)
	(* авария основного осмоса из / блока управления пусками *)
	(* авария резервного осмоса из / блока управлени пусками *)
	(* авария насоса Р03.01/01 *)
	(* *авария основного осмоса по макс давлению датчика РТ03.03/01 *)
	(* *авария основного осмоса по макс давлению датчика РТ03.04/01 *)
	(* PSW336 *)
	(* авария насоса Р03.01/02 *)
	(* авария насоса Р03.02/01 *)
	(* авария насоса Р03.02/02 *)
	(* ошибка блока дозирования Р03.02 *)
	(* авария доз.насоса Н03.04/01, 1=авария *)
	(* авария клапанов 12-14, 1=авария *)
	(* авария доз.насоса Н03.04/02, 1=авария *)
	(* авария клапанов 15-17, 1=авария *)
	(* *авария основного осмоса по макс давлению датчика РТ03.03/02 *)
	(* *авария основного осмоса по макс давлению датчика РТ03.04/02 *)
	(* авария клапана 18, 1=авария *)
	(* PSW337 *)
	#405 PANalarms.0 <= statWordP0301.6
	#406 PANalarms.1 <= statWordP0301.7
	#407 PANalarms.2 <= statWordP0302.6
	#408 PANalarms.3 <= statWordP0302.7
	#409 PANalarms.4 <= DD1_DI_7
	#410 OR(DD1_DI_11, DD1_DI_7, PT030101alarm, PT030201alarm, PT030301alarm, PT030401alarm, QIT030101alarm, FIT030201alarm, FIT030301alarm, P030601alarm)
	#411 osmos1EquipmentAlarm <= #410
	#412 OR(#410, statWordOsmos.6)
	#413 OR(DD1_DI_12, DD1_DI_8, osmos2sensorsAlarm, P030602alarm)
	#414 osmos2EquipmentAlarm <= #413
	#415 OR(statWordOsmos.7, #413)
	#416 AND(#412, #415)
	#417 osmosTotalAlarm <= #416
	#418 PANalarms.5 <= DD1_DI_8
	#419 PANalarms.6 <= P030601alarm
	#420 PANalarms.7 <= P030602alarm
	#421 PANalarms.8 <= DD1_DI_11
	#422 PANalarms.9 <= DD1_DI_12
	#423 PANalarms.10 <= DD1_DI_13
	#424 PANalarms.11 <= dosingErrorP0302
	#425 PANalarms.12 <= osmos1AlarmPT030301
	#426 PANalarms.13 <= osmos1AlarmPT030401
	#427 PANalarms.14 <= osmos2AlarmPT030302
	#428 PANalarms.15 <= osmos2AlarmPT030402
	#429 PANalarms.16 <= FIT0301alarm
	#430 PANalarms.17 <= PT030101alarm
	#431 PANalarms.18 <= PT030201alarm
	#432 PANalarms.19 <= PT030301alarm
	#433 PANalarms.20 <= PT030401alarm
	#434 PANalarms.21 <= QIT030101alarm
	#435 PANalarms.22 <= FIT030201alarm
	#436 PANalarms.23 <= FIT030301alarm
	#437 PANalarms.24 <= PT030102alarm
	#438 PANalarms.25 <= PT030202alarm
	#439 PANalarms.26 <= PT030302alarm
	#440 PANalarms.27 <= PT030402alarm
	#441 PANalarms.28 <= QIT030102alarm
	#442 PANalarms.29 <= FIT030202alarm
	#443 PANalarms.30 <= FIT030302alarm
END_MACRO
#444 MACRO настройка режима запуска осмосов()
	(* работает Р03.01/01 *)
	(* работает Р03.01/02 *)
	(* работает один из насосов Р03.01 *)
	(* *авария основного осмоса по макс давлению датчика РТ03.03/01 *)
	(* *авария основного осмоса по макс давлению датчика РТ03.04/01 *)
	(* *авария резервного осмоса по макс давлению датчика РТ03.03/02 *)
	(* *авария резервного осмоса по макс давлению датчика РТ03.04/02 *)
	#445 OR(statWordP0301.4, statWordP0301.5)
	#446 OR(setWordOsmos.11, osmos1EquipmentAlarm, osmos1AlarmPT030301, osmos1AlarmPT030401)
	#447 OR(setWordOsmos.12, osmos2EquipmentAlarm, osmos2AlarmPT030302, osmos2AlarmPT030402)
	#448 osmosManager:RichTwoPumpManager(#445, setWordOsmos.0, setWordOsmos.1, setWordOsmos.2, setWordOsmos.3, setWordOsmos.4, setWordOsmos.5, setWordOsmos.6, setWordOsmos.7, setWordOsmos.8, setWordOsmos.9, setWordOsmos.10, resetAlarms, DELAY_REPEATED_START_SEC, #446, #447)
	#449 statWordOsmos.0 <= #448.out 1
	#450 statWordOsmos.1 <= #448.out 2
	#451 statWordOsmos.2 <= #448.out 3
	#452 statWordOsmos.3 <= #448.out 4
	#453 counterOsmos1 <= #448.out 5
	#454 counterOsmos2 <= #448.out 6
	#455 daysOfWorkOsmos1 <= #448.out 7
	#456 hoursOfWorkOsmos1 <= #448.out 8
	#457 minutesOfWorkOsmos1 <= #448.out 9
	#458 secondsOfWorkOsmos1 <= #448.out 10
	#459 daysOfWorkOsmos2 <= #448.out 11
	#460 hoursOfWorkOsmos2 <= #448.out 12
	#461 minutesOfWorkOsmos2 <= #448.out 13
	#462 secondsOfWorkOsmos2 <= #448.out 14
	#463 statWordOsmos.4 <= #448.out 15
	#464 statWordOsmos.5 <= #448.out 16
	#465 toNextStartOsmos1timer <= #448.out 17
	#466 toNextStartOsmos2timer <= #448.out 18
	#467 statWordOsmos.6 <= #448.out 19
	#468 statWordOsmos.7 <= #448.out 20
END_MACRO
#469 MACRO передача в панель состояния и наработки осмосов()
	#470 PANstatWordOsmos <= statWordOsmos
	#471 PANdaysOfWorkOsmos1 <= daysOfWorkOsmos1
	#472 PANhoursOfWorkOsmos1 <= hoursOfWorkOsmos1
	#473 PANminutesOfWorkOsmos1 <= minutesOfWorkOsmos1
	#474 PANsecondsOfWorkOsmos1 <= secondsOfWorkOsmos1
	#475 PANtoNextStartOsmos1timer <= toNextStartOsmos1timer
	#476 PANcounterOsmos1 <= counterOsmos1
	#477 PANcounterOsmos2 <= counterOsmos2
	#478 PANdaysOfWorkOsmos2 <= daysOfWorkOsmos2
	#479 PANhoursOfWorkOsmos2 <= hoursOfWorkOsmos2
	#480 PANminutesOfWorkOsmos2 <= minutesOfWorkOsmos2
	#481 PANsecondsOfWorkOsmos2 <= secondsOfWorkOsmos2
	#482 PANtoNextStartOsmos2timer <= toNextStartOsmos2timer
END_MACRO
#483 MACRO алгоритм работы осмосов (насосы Р03.06)()
	(* активен насос Р03.01/02 *)
	(* активен насос Р03.01/01 *)
	(* старт НД03.04/01 *)
	(* пуск основного осмоса *)
	(* клапан 12 *)
	(* клапан 14 *)
	(* клапан 13 *)
	(* клапан 18 *)
	(* активен насос Р03.01/02 *)
	(* активен насос Р03.01/01 *)
	(* старт НД03.04/02 *)
	(* пуск резервного осмоса *)
	(* клапан 15 *)
	(* клапан 17 *)
	(* клапан 16 *)
	(* 0 = уставка расходу своя, не каскад / 1 = уставка каскадная от расхода БМТ *)
	#484 SUB(BMTflowToCascade, FIT0303_SetCascade)
	#485 SEL(isCascade, FIT0303setValue, #484)
	#486 MACRO основной осмос(pin 1 "пуск основного осмоса": statWordOsmos.4, pin 2 "текущие показания датчика РТ03.01/01, МПа": PT030101realValue, pin 3 "уставка датчиков РТ03.01 для старта, МПа": PT0301startValue, pin 4 "активен насос Р03.01/01": statWordP0301.4, pin 5 "активен насос Р03.01/02": statWordP0301.5, pin 6 "текущий расход FIT03,03/01, куб.м/час": FIT030301realValue, pin 7 "заданный расход FIT03,03/01, куб.м/час": #485, pin 8 "КР, расход осн.осм.": KP_F_P030601, pin 9 "I, расход осн.осм.": I_F_P030601, pin 10 "D, расход осн.осм.": D_F_P030601, pin 11 "текущее давление, РТ03.02/01, МПа": PT030201realValue, pin 12 "максимальное давление, РТ03.02/01, МПа": PT0302setMaxValue, pin 13 "КР, давление осн.осм.": KP_P_P030601, pin 14 "I, давление осн.осм.": I_P_P030601, pin 15 "D, давление осн.осм.": D_P_P030601, pin 16 "текущие показания датчика РТ03.03/01, МПа": PT030301realValue, pin 17 "уставка max давление РТ03.03, МПа": PT0303setMaxValue, pin 18 "текущие показания датчика РТ03.04/01, МПа": PT030401realValue, pin 19 "уставка max давление РТ03.04, МПа": PT0304setMaxValue)
		#487 MACRO 1 этап основной осмос(pin 1 "пуск основного осмоса": pin 1)
			#488 OR(pin 1, #495.Q)
			out 2 "клапан 12" <= #488
			#489 tonValve14:TON(IN: pin 1, PT: DELAY_TO_OFF_VALVE)
			#490 OR(#489.Q, #494.Q)
			out 1 "клапан 14/13" <= #490
			out 3 "старт НД03.04/01" <= #491.Q
			out 5 "startP0302" <= #491.Q
			#491 tonValve18:TON(IN: #489.Q, PT: DELAY_TO_OFF_VALVE)
			#492 OR(#491.Q, #493.Q)
			out 4 "клапан 18" <= #492
			#493 tofValve18:TOF(IN: #491.Q, PT: DELAY_TO_CLOSE_VALVE)
			#494 tofValve14:TOF(IN: #493.Q, PT: DELAY_TO_OFF_VALVE)
			#495 tofValve12:TOF(IN: #494.Q, PT: DELAY_TO_OFF_VALVE)
		END_MACRO
		out 7 "клапан 12" <= #487.out 2
		out 11 "старт НД03.04/01" <= #487.out 3
		out 10 "клапан 18" <= #487.out 4
		out 12 "старт доз.насосов Р03.02" <= #487.out 5
		#496 MACRO 2 этап основной осмос(pin 1 "управлять клапанами 13/14": #487.out 1, pin 2 "начать второй этап": #487.out 5, pin 3 "текущие показания датчика РТ03.01/01": pin 2, pin 4 "уставка датчиков РТ03.01 для старта": pin 3, pin 5 "активен насос Р03.01/01": pin 4, pin 6 "активен насос Р03.01/02": pin 5)
			#497 +(DELAY_TO_SWITCH_VALVE, DELAY_TO_CLOSE_VALVE)
			#498 tonSwitchValve1413:TON(IN: #502, PT: DELAY_TO_SWITCH_VALVE)
			#499 HoldingToEndProcValve:TOF(IN: #498.Q, PT: #497)
			#500 SEL(#499.Q, pin 1, #504.Q)
			out 1 "клапан 14" <= #500
			#501 >(pin 3, pin 4)
			#502 AND(#501, #505.Q)
			out 5 "пуск насоса Р03.06/01" <= #502
			#503 valve1413switcher:IfBOOL(key: #499.Q, input: pin 1)
			#504 delayToSwitchValve14to13:TOF(IN: #503.keyFALSE, PT: DELAY_TO_OFF_VALVE)
			out 2 "клапан 13" <= #503.keyTRUE
			#505 tonPT030101:TON(IN: pin 2, PT: DELAY_TO_CHECK_PT0301)
			#506 AND(pin 5, #507)
			out 3 "авария насоса Р03.01/01" <= #506
			#507 AND(#505.Q, #508)
			#508 <(pin 3, pin 4)
			#509 AND(#507, pin 6)
			out 4 "авария насоса Р03.01/ 02" <= #509
		END_MACRO
		out 9 "клапан 14" <= #496.out 1
		out 8 "клапан 13" <= #496.out 2
		out 13 "авария низкое давление насос Р03.01/01" <= #496.out 3
		out 14 "авария низкое давление насос Р03.01/02" <= #496.out 4
		out 1 "пуск насоса Р03.06/01" <= #496.out 5
		#510 AND(#496.out 5, #511)
		out 2 "авария осмос 1  макс.давл.РТ03.03/01" <= #510
		#511 >=(pin 16, pin 17)
		#512 AND(#496.out 5, #513)
		out 3 "авария осмос 1  макс.давл.РТ03.04/01" <= #512
		#513 >=(pin 18, pin 19)
		#514 MACRO управление производительностью Р03.06/01(pin 1 "текущий расход, FIT03.03/01, куб.м/час": pin 6, pin 2 "заданный расход, FIT03.03/01 , куб.м/час": pin 7, pin 3 "КР, расход": pin 8, pin 4 "I, сек, расход": pin 9, pin 5 "D, сек, расход": pin 10, pin 6 "текущее давление, РТ03.02/01, МПа": pin 11, pin 7 "максимальное давление, РТ03.02/01, МПа": pin 12, pin 8 "КР, давление": pin 13, pin 9 "I, сек, давление": pin 14, pin 10 "D, сек, давление": pin 15)
			(* Задача: поддерживать заданный расход. / Если давление при этом превысит заданный уровень, / снижать производительность, не глядя на расход. / В идеале два ПИД-регулятора ПЛАВНО передают управление друг-другу. / Если реальность оказалась более сурова и регуляторы мешают друг другу, / то есть два пути: / 1. Настраивать ПИД-регуляторы коэффициентами / 2. Переосмысливать и переделывать этот блок. *)
			(* tесли выход менььше нуля, то ноль, / иначе - то, что насчитали *)
			#515 F_P030601:PID(ACTUAL: pin 1, SET_POINT: pin 2, KP: pin 3, TN: pin 4, TV: pin 5, Y_MANUAL: -, Y_OFFSET: -, Y_MIN: 0, Y_MAX: 100, MANUAL: -, RESET: #515.OVERFLOW)
			out 1 "производительность по расходу, 0...100%" <= #515.Y
			#516 <(#518, 0)
			#517 SEL(#516, #518, 0)
			out 3 "производительность итог, 0...100%" <= #517
			#518 -(#515.Y, #519)
			#519 -(100, #520.Y)
			out 2 "коррекция по давлению, 0...100%" <= #519
			#520 P_P030601:PID(ACTUAL: pin 6, SET_POINT: pin 7, KP: pin 8, TN: pin 9, TV: pin 10, Y_MANUAL: -, Y_OFFSET: -, Y_MIN: 0, Y_MAX: 100, MANUAL: -, RESET: #520.OVERFLOW)
		END_MACRO
		out 4 "производительность по расходу осн.осмос, 0...100%" <= #514.out 1
		out 5 "коррекция по давлению осн.осмос, 0...100%" <= #514.out 2
		out 6 "производительность итог осн.осмос, 0...100%" <= #514.out 3
	END_MACRO
	#521 P030601start <= #486.out 1
	#522 osmos1AlarmPT030301 <= #486.out 2
	#523 osmos1AlarmPT030401 <= #486.out 3
	#524 Yout_F_P030601 <= #486.out 4
	#525 Yout_P_P030601 <= #486.out 5
	#526 Yout_Total_P030601 <= #486.out 6
	#527 DD1_DO_6 <= #486.out 7
	#528 DD1_DO_7 <= #486.out 8
	#529 DD1_DO_8 <= #486.out 9
	#530 DD1_DO_4 <= #486.out 11
	#531 lowPT030101_P030101 <= #486.out 13
	#532 lowPT030101_P030102 <= #486.out 14
	#533 MACRO резервный осмос(pin 1 "пуск резервного осмоса": statWordOsmos.5, pin 2 "текущие показания РТ01.03/02": PT030102realValue, pin 3 "уставка РТ03.01/02 для старта": PT0301startValue, pin 4 "активен насос Р03.01/01": statWordP0301.4, pin 5 "активен насос Р03.01/02": statWordP0301.5, pin 6 "текущий расход, FIT03/03/02, куб.м/час": FIT030302realValue, pin 7 "заданный расход, FIT03/03/02, куб.м/час": #485, pin 8 "KP, расход, осмос 2": KP_F_P030602, pin 9 "I, расход, осмос 2": I_F_P030602, pin 10 "D, расход, осмос 2": D_F_P030602, pin 11 "текущее давление PT03.02/02, МПа": PT030202realValue, pin 12 "максимальное давление PT03.02/02, МПа": PT0302setMaxValue, pin 13 "KP, давление, осмос 2": KP_P_P030602, pin 14 "I, давление, осмос 2": I_P_P030602, pin 15 "D, давление, осмос 2": D_P_P030602, pin 16 "текущее давление РТ03.03/02": PT030302realValue, pin 17 "задание max давление РТ03.03/02": PT0303setMaxValue, pin 18 "текущее давление РТ03.04/02": PT030402realValue, pin 19 "задание max давление РТ03.04/02": PT0304setMaxValue)
		#534 MACRO 1 этап резервный осмос(pin 1 "пуск резервного осмоса": pin 1)
			#535 OR(pin 1, #542.Q)
			out 2 "клапан 15" <= #535
			#536 tonValve17:TON(IN: pin 1, PT: DELAY_TO_OFF_VALVE)
			#537 OR(#536.Q, #541.Q)
			out 1 "клапан 16/17" <= #537
			out 3 "старт НД03.04/02" <= #538.Q
			out 5 "startP0302" <= #538.Q
			#538 tonValve18rez:TON(IN: #536.Q, PT: DELAY_TO_OFF_VALVE)
			#539 OR(#538.Q, #540.Q)
			out 4 "клапан 18" <= #539
			#540 tofValve18rez:TOF(IN: #538.Q, PT: DELAY_TO_CLOSE_VALVE)
			#541 tofValve17:TOF(IN: #540.Q, PT: DELAY_TO_OFF_VALVE)
			#542 tofValve15:TOF(IN: #541.Q, PT: DELAY_TO_OFF_VALVE)
		END_MACRO
		out 5 "клапан 15" <= #534.out 2
		out 6 "старт НД03.04/02" <= #534.out 3
		out 2 "клапан 18" <= #534.out 4
		out 1 "пуск Р0302" <= #534.out 5
		#543 MACRO 2 этап резервный осмос(pin 1 "управлять клапанами 16/17": #534.out 1, pin 2 "начать второй этап": #534.out 5, pin 3 "текущие показания датчика РТ03.01/02": pin 2, pin 4 "уставка датчиков РТ03.01 для старта": pin 3, pin 5 "активен насос Р03.01/01": pin 4, pin 6 "активен насос Р03.01/02": pin 5)
			#544 +(DELAY_TO_SWITCH_VALVE, DELAY_TO_CLOSE_VALVE)
			#545 tonSwitchValve1716:TON(IN: #549, PT: DELAY_TO_SWITCH_VALVE)
			#546 HoldingToEndProcValveRez:TOF(IN: #545.Q, PT: #544)
			#547 SEL(#546.Q, pin 1, #551.Q)
			out 1 "клапан 17" <= #547
			#548 >(pin 3, pin 4)
			#549 AND(#548, #552.Q)
			out 5 "пуск насоса Р03.06/02" <= #549
			#550 valve1716switcher:IfBOOL(key: #546.Q, input: pin 1)
			#551 delayToSwitchValve17to16:TOF(IN: #550.keyFALSE, PT: DELAY_TO_OFF_VALVE)
			out 2 "клапан 16" <= #550.keyTRUE
			#552 tonPT030102:TON(IN: pin 2, PT: DELAY_TO_CHECK_PT0301)
			#553 AND(pin 5, #554)
			out 3 "авария насоса Р03.01/01" <= #553
			#554 AND(#552.Q, #555)
			#555 <(pin 3, pin 4)
			#556 AND(#554, pin 6)
			out 4 "авария насоса Р03.01/ 02" <= #556
		END_MACRO
		out 3 "клапан 17" <= #543.out 1
		out 4 "клапан 16" <= #543.out 2
		out 7 "авария низкое давление насос Р03.03/01" <= #543.out 3
		out 8 "авария низкое давление насос Р03.03/02" <= #543.out 4
		out 9 "пуск насоса Р03.06/02" <= #543.out 5
		#557 AND(#543.out 5, #558)
		out 13 "авария осмос 2 max давление РТ03.03/02" <= #557
		#558 >=(pin 16, pin 17)
		#559 AND(#543.out 5, #560)
		out 14 "авария осмос 2 max давление РТ03.04/02" <= #559
		#560 >=(pin 18, pin 19)
		#561 MACRO управление производительностью Р03.06/02(pin 1 "текущий расход, FIT03.03/02, куб.м/час": pin 6, pin 2 "заданный расход, FIT03.03/02 , куб.м/час": pin 7, pin 3 "КР, расход, осмос 2": pin 8, pin 4 "I, сек, расход, осмос 2": pin 9, pin 5 "D, сек, расход, осмос 2": pin 10, pin 6 "текущее давление, РТ03.02/02, МПа": pin 11, pin 7 "максимальное давление, РТ03.02/02, МПа": pin 12, pin 8 "КР, давление, осмос 2": pin 13, pin 9 "I, сек, давление, осмос 2": pin 14, pin 10 "D, сек, давление, осмос 2": pin 15)
			(* Задача: поддерживать заданный расход. / Если давление при этом превысит заданный уровень, / снижать производительность, не глядя на расход. / В идеале два ПИД-регулятора ПЛАВНО передают управление друг-другу. / Если реальность оказалась более сурова и регуляторы мешают друг другу, / то есть два пути: / 1. Настраивать ПИД-регуляторы коэффициентами / 2. Переосмысливать и переделывать этот блок. *)
			(* tесли выход менььше нуля, то ноль, / иначе - то, что насчитали *)
			#562 F_P030602:PID(ACTUAL: pin 1, SET_POINT: pin 2, KP: pin 3, TN: pin 4, TV: pin 5, Y_MANUAL: -, Y_OFFSET: -, Y_MIN: 0, Y_MAX: 100, MANUAL: -, RESET: #562.OVERFLOW)
			out 1 "производительность по расходу, 0...100%" <= #562.Y
			#563 <(#565, 0)
			#564 SEL(#563, #565, 0)
			out 3 "производительность итог, 0...100%" <= #564
			#565 -(#562.Y, #566)
			#566 -(100, #567.Y)
			out 2 "коррекция по давлению, 0...100%" <= #566
			#567 P_P030602:PID(ACTUAL: pin 6, SET_POINT: pin 7, KP: pin 8, TN: pin 9, TV: pin 10, Y_MANUAL: -, Y_OFFSET: -, Y_MIN: 0, Y_MAX: 100, MANUAL: -, RESET: #567.OVERFLOW)
		END_MACRO
		out 10 "производительность по расходу, рез.осмос, 0...100%" <= #561.out 1
		out 11 "коррекция по давлению, рез.осмос, 0...100%" <= #561.out 2
		out 12 "производительность итог, 0...100%" <= #561.out 3
	END_MACRO
	#568 DD1_DO_11 <= #533.out 3
	#569 DD1_DO_10 <= #533.out 4
	#570 DD1_DO_9 <= #533.out 5
	#571 DD1_DO_5 <= #533.out 6
	#572 lowPT030102_P030101 <= #533.out 7
	#573 lowPT030102_P030102 <= #533.out 8
	#574 P030602start <= #533.out 9
	#575 Yout_F_P030602 <= #533.out 10
	#576 Yout_P_P030602 <= #533.out 11
	#577 Yout_Total_P030602 <= #533.out 12
	#578 osmos2AlarmPT030302 <= #533.out 13
	#579 osmos2AlarmPT030402 <= #533.out 14
	#580 OR(#486.out 10, #533.out 2)
	#581 DD1_DO_1 <= #580
	#582 OR(#486.out 12, #533.out 1)
	#583 startP0302 <= #582
END_MACRO
#584 MACRO передача наработки и состояния доз.насоса Р03.02 в панель()
	#585 PANstatWordP0302 <= statWordP0302
	#586 PANdaysOfWorkP030201 <= daysOfWorkP030201
	#587 PANhoursOfWorkP030201 <= hoursOfWorkP030201
	#588 PANminutesOfWorkP030201 <= minutesOfWorkP030201
	#589 PANsecondsOfWorkP030201 <= secondsOfWorkP030201
	#590 PANtoNextStartP030201timer <= toNextStartP030201timer
	#591 PANcounterP030201 <= counterP030201
	#592 PANdaysOfWorkP030202 <= daysOfWorkP030202
	#593 PANhoursOfWorkP030202 <= hoursOfWorkP030202
	#594 PANminutesOfWorkP030202 <= minutesOfWorkP030202
	#595 PANsecondsOfWorkP030202 <= secondsOfWorkP030202
	#596 PANtoNextStartP030202timer <= toNextStartP030202timer
	#597 PANcounterP030202 <= counterP030202
END_MACRO
#598 WORD_TO_BOOL(PANsetWordP0302)
#599 tof3:TOF(IN: #598, PT: T#1s)
#600 MOVE(EN: #599.Q, PANsetWordP0302)
#601 setWordP0302 <= #600
#602 WORD_TO_BOOL(OPANsetWordP0302)
#603 tof4:TOF(IN: #602, PT: T#1s)
#604 OR(#599.Q, #603.Q)
#605 MOVE(EN: #604, statWordP0302)
#606 setWordP0302onStart <= #605
#607 MOVE(EN: #603.Q, OPANsetWordP0302)
#608 setWordP0302 <= #607
#609 WORD_TO_BOOL(PANsetWordOsmos)
#610 tof5:TOF(IN: #609, PT: T#1s)
#611 MOVE(EN: #610.Q, PANsetWordOsmos)
#612 setWordOsmos <= #611
#613 WORD_TO_BOOL(OPANsetWordOsmos)
#614 tof6:TOF(IN: #613, PT: T#1s)
#615 OR(#610.Q, #614.Q)
#616 MOVE(EN: #615, statWordOsmos)
#617 setWordOsmosOnStart <= #616
#618 MOVE(EN: #614.Q, OPANsetWordOsmos)
#619 setWordOsmos <= #618
_END_CFC_
END_PROGRAM
